gfCNCPoint2[18031] = {X 270.1696, Y 41.5937, Z -3.0000, A 0.000, B 0.000, C 0.000 }
gfCNCPoint2[18032] = {X 270.6458, Y 42.3821, Z -3.0000, A 0.000, B 0.000, C 0.000 }
gfCNCPoint2[18033] = {X 270.9441, Y 43.2536, Z -3.0000, A 0.000, B 0.000, C 0.000 }
gfCNCPoint2[18034] = {X 271.0508, Y 44.1686, Z -3.0000, A 0.000, B 0.000, C 0.000 }
gfCNCPoint2[18035] = {X 271.0510, Y 45.0000, Z -3.0000, A 0.000, B 0.000, C 0.000 }
gfCNCPoint2[18036] = {X 270.9427, Y 45.9613, Z -3.0000, A 0.000, B 0.000, C 0.000 }
gfCNCPoint2[18037] = {X 270.6232, Y 46.8744, Z -3.0000, A 0.000, B 0.000, C 0.000 }
gfCNCPoint2[18038] = {X 270.1085, Y 47.6935, Z -3.0000, A 0.000, B 0.000, C 0.000 }
gfCNCPoint2[18039] = {X 269.4245, Y 48.3775, Z -3.0000, A 0.000, B 0.000, C 0.000 }
gfCNCPoint2[18040] = {X 268.6054, Y 48.8922, Z -3.0000, A 0.000, B 0.000, C 0.000 }
gfCNCPoint2[18041] = {X 267.6923, Y 49.2117, Z -3.0000, A 0.000, B 0.000, C 0.000 }
gfCNCPoint2[18042] = {X 266.7310, Y 49.3200, Z -3.0000, A 0.000, B 0.000, C 0.000 }
gfCNCPoint2[18043] = {X 260.2876, Y 49.3200, Z -3.0000, A 0.000, B 0.000, C 0.000 }
gfCNCPoint2[18044] = {X 259.3310, Y 49.2128, Z -3.0000, A 0.000, B 0.000, C 0.000 }
gfCNCPoint2[18045] = {X 258.4219, Y 48.8963, Z -3.0000, A 0.000, B 0.000, C 0.000 }
gfCNCPoint2[18046] = {X 257.6054, Y 48.3865, Z -3.0000, A 0.000, B 0.000, C 0.000 }
gfCNCPoint2[18047] = {X 256.9221, Y 47.7085, Z -3.0000, A 0.000, B 0.000, C 0.000 }
gfCNCPoint2[18048] = {X 256.4059, Y 46.8960, Z -3.0000, A 0.000, B 0.000, C 0.000 }
gfCNCPoint2[18049] = {X 256.0824, Y 45.9894, Z -3.0000, A 0.000, B 0.000, C 0.000 }
gfCNCPoint2[18050] = {X 255.9677, Y 45.0336, Z -3.0000, A 0.000, B 0.000, C 0.000 }
gfCNCPoint2[18051] = {X 255.9680, Y 44.1494, Z -3.0000, A 0.000, B 0.000, C 0.000 }
gfCNCPoint2[18052] = {X 256.0784, Y 43.2364, Z -3.0000, A 0.000, B 0.000, C 0.000 }
gfCNCPoint2[18053] = {X 256.3796, Y 42.3675, Z -3.0000, A 0.000, B 0.000, C 0.000 }
gfCNCPoint2[18054] = {X 256.8579, Y 41.5821, Z -3.0000, A 0.000, B 0.000, C 0.000 }
gfCNCPoint2[18055] = {X 257.4915, Y 40.9157, Z -3.0000, A 0.000, B 0.000, C 0.000 }
gfCNCPoint2[18056] = {X 257.4915, Y 34.4738, Z -3.0000, A 0.000, B 0.000, C 0.000 }
gfCNCPoint2[18057] = {X 254.7671, Y 34.4738, Z -3.0000, A 0.000, B 0.000, C 0.000 }
gfCNCPoint2[18058] = {X 250.4836, Y 42.8182, Z -3.0000, A 0.000, B 0.000, C 0.000 }
gfCNCPoint2[18059] = {X 250.6527, Y 43.4861, Z -3.0000, A 0.000, B 0.000, C 0.000 }
gfCNCPoint2[18060] = {X 250.7134, Y 44.1723, Z -3.0000, A 0.000, B 0.000, C 0.000 }
gfCNCPoint2[18061] = {X 250.7136, Y 45.0000, Z -3.0000, A 0.000, B 0.000, C 0.000 }
gfCNCPoint2[18062] = {X 250.6052, Y 45.9613, Z -3.0000, A 0.000, B 0.000, C 0.000 }
gfCNCPoint2[18063] = {X 250.2857, Y 46.8744, Z -3.0000, A 0.000, B 0.000, C 0.000 }
gfCNCPoint2[18064] = {X 249.7711, Y 47.6935, Z -3.0000, A 0.000, B 0.000, C 0.000 }
gfCNCPoint2[18065] = {X 249.0870, Y 48.3775, Z -3.0000, A 0.000, B 0.000, C 0.000 }
gfCNCPoint2[18066] = {X 248.2679, Y 48.8922, Z -3.0000, A 0.000, B 0.000, C 0.000 }
gfCNCPoint2[18067] = {X 247.3548, Y 49.2117, Z -3.0000, A 0.000, B 0.000, C 0.000 }
gfCNCPoint2[18068] = {X 246.3936, Y 49.3200, Z -3.0000, A 0.000, B 0.000, C 0.000 }
gfCNCPoint2[18069] = {X 239.8075, Y 49.3200, Z -3.0000, A 0.000, B 0.000, C 0.000 }
gfCNCPoint2[18070] = {X 238.8462, Y 49.2117, Z -3.0000, A 0.000, B 0.000, C 0.000 }
gfCNCPoint2[18071] = {X 237.9331, Y 48.8922, Z -3.0000, A 0.000, B 0.000, C 0.000 }
gfCNCPoint2[18072] = {X 237.1141, Y 48.3775, Z -3.0000, A 0.000, B 0.000, C 0.000 }
gfCNCPoint2[18073] = {X 236.4300, Y 47.6935, Z -3.0000, A 0.000, B 0.000, C 0.000 }
gfCNCPoint2[18074] = {X 235.9153, Y 46.8745, Z -3.0000, A 0.000, B 0.000, C 0.000 }
gfCNCPoint2[18075] = {X 235.5958, Y 45.9614, Z -3.0000, A 0.000, B 0.000, C 0.000 }
gfCNCPoint2[18076] = {X 235.4875, Y 45.0001, Z -3.0000, A 0.000, B 0.000, C 0.000 }
gfCNCPoint2[18077] = {X 235.4879, Y 44.1494, Z -3.0000, A 0.000, B 0.000, C 0.000 }
gfCNCPoint2[18078] = {X 235.5856, Y 43.2935, Z -3.0000, A 0.000, B 0.000, C 0.000 }
gfCNCPoint2[18079] = {X 235.8511, Y 42.4740, Z -3.0000, A 0.000, B 0.000, C 0.000 }
gfCNCPoint2[18080] = {X 236.2739, Y 41.7236, Z -3.0000, A 0.000, B 0.000, C 0.000 }
gfCNCPoint2[18081] = {X 236.8373, Y 41.0719, Z -3.0000, A 0.000, B 0.000, C 0.000 }
gfCNCPoint2[18082] = {X 237.5187, Y 40.5449, Z -3.0000, A 0.000, B 0.000, C 0.000 }
gfCNCPoint2[18083] = {X 238.2911, Y 40.1637, Z -3.0000, A 0.000, B 0.000, C 0.000 }
gfCNCPoint2[18084] = {X 242.2805, Y 32.3549, Z -3.0000, A 0.000, B 0.000, C 0.000 }
gfCNCPoint2[18085] = {X 241.1106, Y 31.5686, Z -3.0000, A 0.000, B 0.000, C 0.000 }
gfCNCPoint2[18086] = {X 240.0474, Y 30.6429, Z -3.0000, A 0.000, B 0.000, C 0.000 }
gfCNCPoint2[18087] = {X 239.1077, Y 29.5922, Z -3.0000, A 0.000, B 0.000, C 0.000 }
gfCNCPoint2[18088] = {X 238.3058, Y 28.4329, Z -3.0000, A 0.000, B 0.000, C 0.000 }
gfCNCPoint2[18089] = {X 237.6543, Y 27.1828, Z -3.0000, A 0.000, B 0.000, C 0.000 }
gfCNCPoint2[18090] = {X 237.1633, Y 25.8614, Z -3.0000, A 0.000, B 0.000, C 0.000 }
gfCNCPoint2[18091] = {X 236.7431, Y 24.0500, Z -3.0000, A 0.000, B 0.000, C 0.000 }
gfCNCPoint2[18092] = {X 236.5290, Y 22.2028, Z -3.0000, A 0.000, B 0.000, C 0.000 }
gfCNCPoint2[18093] = {X 236.5236, Y 20.3432, Z -3.0000, A 0.000, B 0.000, C 0.000 }
gfCNCPoint2[18094] = {X 236.7271, Y 18.4949, Z -3.0000, A 0.000, B 0.000, C 0.000 }
gfCNCPoint2[18095] = {X 237.1368, Y 16.6810, Z -3.0000, A 0.000, B 0.000, C 0.000 }
gfCNCPoint2[18096] = {X 237.7071, Y 15.1054, Z -3.0000, A 0.000, B 0.000, C 0.000 }
gfCNCPoint2[18097] = {X 238.4940, Y 13.6260, Z -3.0000, A 0.000, B 0.000, C 0.000 }
gfCNCPoint2[18098] = {X 239.4818, Y 12.2725, Z -3.0000, A 0.000, B 0.000, C 0.000 }
gfCNCPoint2[18099] = {X 240.6507, Y 11.0718, Z -3.0000, A 0.000, B 0.000, C 0.000 }
gfCNCPoint2[18100] = {X 241.9772, Y 10.0481, Z -3.0000, A 0.000, B 0.000, C 0.000 }
gfCNCPoint2[18101] = {X 243.4350, Y 9.2218, Z -3.0000, A 0.000, B 0.000, C 0.000 }
gfCNCPoint2[18102] = {X 244.9947, Y 8.6094, Z -3.0000, A 0.000, B 0.000, C 0.000 }
gfCNCPoint2[18103] = {X 246.6252, Y 8.2232, Z -3.0000, A 0.000, B 0.000, C 0.000 }
gfCNCPoint2[18104] = {X 248.7221, Y 7.9518, Z -3.0000, A 0.000, B 0.000, C 0.000 }
gfCNCPoint2[18105] = {X 250.8350, Y 7.8712, Z -3.0000, A 0.000, B 0.000, C 0.000 }
gfCNCPoint2[18106] = {X 266.7634, Y 7.8712, Z -3.0000, A 0.000, B 0.000, C 0.000 }
gfCNCPoint2[18107] = {X 267.7184, Y 7.9860, Z -3.0000, A 0.000, B 0.000, C 0.000 }
gfCNCPoint2[18108] = {X 268.6245, Y 8.3091, Z -3.0000, A 0.000, B 0.000, C 0.000 }
gfCNCPoint2[18109] = {X 269.4366, Y 8.8247, Z -3.0000, A 0.000, B 0.000, C 0.000 }
gfCNCPoint2[18110] = {X 270.1147, Y 9.5070, Z -3.0000, A 0.000, B 0.000, C 0.000 }
gfCNCPoint2[18111] = {X 270.6250, Y 10.3225, Z -3.0000, A 0.000, B 0.000, C 0.000 }
gfCNCPoint2[18112] = {X 270.9424, Y 11.2305, Z -3.0000, A 0.000, B 0.000, C 0.000 }
gfCNCPoint2[18113] = {X 271.0510, Y 12.1863, Z -3.0000, A 0.000, B 0.000, C 0.000 }
gfCNCPoint2[18114] = {X 271.0508, Y 13.0225, Z -3.0000, A 0.000, B 0.000, C 0.000 }
gfCNCPoint2[18115] = {X 270.9424, Y 13.9406, Z -3.0000, A 0.000, B 0.000, C 0.000 }
gfCNCPoint2[18116] = {X 270.6412, Y 14.8147, Z -3.0000, A 0.000, B 0.000, C 0.000 }
gfCNCPoint2[18117] = {X 270.1608, Y 15.6046, Z -3.0000, A 0.000, B 0.000, C 0.000 }
gfCNCPoint2[18118] = {X 269.5234, Y 16.2742, Z -3.0000, A 0.000, B 0.000, C 0.000 }
gfCNCPoint2[18119] = {X 269.5233, Y 28.5936, Z -3.0000, A 0.000, B 0.000, C 0.000 }
gfCNCPoint2[18120] = {X 273.5233, Y 28.5937, Z -3.0000, A 0.000, B 0.000, C 0.000 }
gfCNCPoint2[18121] = {X 269.4433, Y 28.5936, Z -3.0000, A 0.000, B 0.000, C 0.000 }
gfCNCPoint2[18122] = {X 269.4432, Y 40.9513, Z -3.0000, A 0.000, B 0.000, C 0.000 }
gfCNCPoint2[18123] = {X 269.4859, Y 40.9857, Z -3.0000, A 0.000, B 0.000, C 0.000 }
gfCNCPoint2[18124] = {X 270.1064, Y 41.6428, Z -3.0000, A 0.000, B 0.000, C 0.000 }
gfCNCPoint2[18125] = {X 270.5736, Y 42.4165, Z -3.0000, A 0.000, B 0.000, C 0.000 }
gfCNCPoint2[18126] = {X 270.8662, Y 43.2716, Z -3.0000, A 0.000, B 0.000, C 0.000 }
gfCNCPoint2[18127] = {X 270.9708, Y 44.1693, Z -3.0000, A 0.000, B 0.000, C 0.000 }
gfCNCPoint2[18128] = {X 270.9710, Y 45.0000, Z -3.0000, A 0.000, B 0.000, C 0.000 }
gfCNCPoint2[18129] = {X 270.8647, Y 45.9435, Z -3.0000, A 0.000, B 0.000, C 0.000 }
gfCNCPoint2[18130] = {X 270.5511, Y 46.8397, Z -3.0000, A 0.000, B 0.000, C 0.000 }
gfCNCPoint2[18131] = {X 270.0460, Y 47.6436, Z -3.0000, A 0.000, B 0.000, C 0.000 }
gfCNCPoint2[18132] = {X 269.3746, Y 48.3150, Z -3.0000, A 0.000, B 0.000, C 0.000 }
gfCNCPoint2[18133] = {X 268.5707, Y 48.8201, Z -3.0000, A 0.000, B 0.000, C 0.000 }
gfCNCPoint2[18134] = {X 267.6745, Y 49.1337, Z -3.0000, A 0.000, B 0.000, C 0.000 }
gfCNCPoint2[18135] = {X 266.7310, Y 49.2400, Z -3.0000, A 0.000, B 0.000, C 0.000 }
gfCNCPoint2[18136] = {X 260.2876, Y 49.2400, Z -3.0000, A 0.000, B 0.000, C 0.000 }
gfCNCPoint2[18137] = {X 259.3487, Y 49.1347, Z -3.0000, A 0.000, B 0.000, C 0.000 }
gfCNCPoint2[18138] = {X 258.4564, Y 48.8242, Z -3.0000, A 0.000, B 0.000, C 0.000 }
gfCNCPoint2[18139] = {X 257.6550, Y 48.3238, Z -3.0000, A 0.000, B 0.000, C 0.000 }
gfCNCPoint2[18140] = {X 256.9844, Y 47.6583, Z -3.0000, A 0.000, B 0.000, C 0.000 }
gfCNCPoint2[18141] = {X 256.4777, Y 46.8609, Z -3.0000, A 0.000, B 0.000, C 0.000 }
gfCNCPoint2[18142] = {X 256.1603, Y 45.9711, Z -3.0000, A 0.000, B 0.000, C 0.000 }
gfCNCPoint2[18143] = {X 256.0477, Y 45.0330, Z -3.0000, A 0.000, B 0.000, C 0.000 }
gfCNCPoint2[18144] = {X 256.0480, Y 44.1505, Z -3.0000, A 0.000, B 0.000, C 0.000 }
gfCNCPoint2[18145] = {X 256.1585, Y 43.2454, Z -3.0000, A 0.000, B 0.000, C 0.000 }
gfCNCPoint2[18146] = {X 256.4599, Y 42.3850, Z -3.0000, A 0.000, B 0.000, C 0.000 }
gfCNCPoint2[18147] = {X 256.9383, Y 41.6088, Z -3.0000, A 0.000, B 0.000, C 0.000 }
gfCNCPoint2[18148] = {X 257.5715, Y 40.9529, Z -3.0000, A 0.000, B 0.000, C 0.000 }
gfCNCPoint2[18149] = {X 257.5715, Y 34.3938, Z -3.0000, A 0.000, B 0.000, C 0.000 }
gfCNCPoint2[18150] = {X 254.7182, Y 34.3938, Z -3.0000, A 0.000, B 0.000, C 0.000 }
gfCNCPoint2[18151] = {X 250.3969, Y 42.8120, Z -3.0000, A 0.000, B 0.000, C 0.000 }
gfCNCPoint2[18152] = {X 250.5709, Y 43.4828, Z -3.0000, A 0.000, B 0.000, C 0.000 }
gfCNCPoint2[18153] = {X 250.6334, Y 44.1730, Z -3.0000, A 0.000, B 0.000, C 0.000 }
gfCNCPoint2[18154] = {X 250.6336, Y 45.0000, Z -3.0000, A 0.000, B 0.000, C 0.000 }
gfCNCPoint2[18155] = {X 250.5273, Y 45.9435, Z -3.0000, A 0.000, B 0.000, C 0.000 }
gfCNCPoint2[18156] = {X 250.2137, Y 46.8397, Z -3.0000, A 0.000, B 0.000, C 0.000 }
gfCNCPoint2[18157] = {X 249.7085, Y 47.6436, Z -3.0000, A 0.000, B 0.000, C 0.000 }
gfCNCPoint2[18158] = {X 249.0372, Y 48.3150, Z -3.0000, A 0.000, B 0.000, C 0.000 }
gfCNCPoint2[18159] = {X 248.2332, Y 48.8201, Z -3.0000, A 0.000, B 0.000, C 0.000 }
gfCNCPoint2[18160] = {X 247.3370, Y 49.1337, Z -3.0000, A 0.000, B 0.000, C 0.000 }
gfCNCPoint2[18161] = {X 246.3936, Y 49.2400, Z -3.0000, A 0.000, B 0.000, C 0.000 }
gfCNCPoint2[18162] = {X 239.8075, Y 49.2400, Z -3.0000, A 0.000, B 0.000, C 0.000 }
gfCNCPoint2[18163] = {X 238.8640, Y 49.1337, Z -3.0000, A 0.000, B 0.000, C 0.000 }
gfCNCPoint2[18164] = {X 237.9679, Y 48.8201, Z -3.0000, A 0.000, B 0.000, C 0.000 }
gfCNCPoint2[18165] = {X 237.1639, Y 48.3150, Z -3.0000, A 0.000, B 0.000, C 0.000 }
gfCNCPoint2[18166] = {X 236.4926, Y 47.6436, Z -3.0000, A 0.000, B 0.000, C 0.000 }
gfCNCPoint2[18167] = {X 235.9874, Y 46.8397, Z -3.0000, A 0.000, B 0.000, C 0.000 }
gfCNCPoint2[18168] = {X 235.6738, Y 45.9436, Z -3.0000, A 0.000, B 0.000, C 0.000 }
gfCNCPoint2[18169] = {X 235.5675, Y 45.0001, Z -3.0000, A 0.000, B 0.000, C 0.000 }
gfCNCPoint2[18170] = {X 235.5679, Y 44.1505, Z -3.0000, A 0.000, B 0.000, C 0.000 }
gfCNCPoint2[18171] = {X 235.6649, Y 43.3054, Z -3.0000, A 0.000, B 0.000, C 0.000 }
gfCNCPoint2[18172] = {X 235.9285, Y 42.4967, Z -3.0000, A 0.000, B 0.000, C 0.000 }
gfCNCPoint2[18173] = {X 236.3483, Y 41.7570, Z -3.0000, A 0.000, B 0.000, C 0.000 }
gfCNCPoint2[18174] = {X 236.9073, Y 41.1159, Z -3.0000, A 0.000, B 0.000, C 0.000 }
gfCNCPoint2[18175] = {X 237.5830, Y 40.5992, Z -3.0000, A 0.000, B 0.000, C 0.000 }
gfCNCPoint2[18176] = {X 238.3482, Y 40.2278, Z -3.0000, A 0.000, B 0.000, C 0.000 }
gfCNCPoint2[18177] = {X 242.3863, Y 32.3238, Z -3.0000, A 0.000, B 0.000, C 0.000 }
gfCNCPoint2[18178] = {X 241.2093, Y 31.5432, Z -3.0000, A 0.000, B 0.000, C 0.000 }
gfCNCPoint2[18179] = {X 240.1396, Y 30.6212, Z -3.0000, A 0.000, B 0.000, C 0.000 }
gfCNCPoint2[18180] = {X 239.1939, Y 29.5723, Z -3.0000, A 0.000, B 0.000, C 0.000 }
gfCNCPoint2[18181] = {X 238.3873, Y 28.4131, Z -3.0000, A 0.000, B 0.000, C 0.000 }
gfCNCPoint2[18182] = {X 237.7325, Y 27.1618, Z -3.0000, A 0.000, B 0.000, C 0.000 }
gfCNCPoint2[18183] = {X 237.2398, Y 25.8383, Z -3.0000, A 0.000, B 0.000, C 0.000 }
gfCNCPoint2[18184] = {X 236.8218, Y 24.0357, Z -3.0000, A 0.000, B 0.000, C 0.000 }
gfCNCPoint2[18185] = {X 236.6088, Y 22.1976, Z -3.0000, A 0.000, B 0.000, C 0.000 }
gfCNCPoint2[18186] = {X 236.6035, Y 20.3472, Z -3.0000, A 0.000, B 0.000, C 0.000 }
gfCNCPoint2[18187] = {X 236.8060, Y 18.5079, Z -3.0000, A 0.000, B 0.000, C 0.000 }
gfCNCPoint2[18188] = {X 237.2138, Y 16.7029, Z -3.0000, A 0.000, B 0.000, C 0.000 }
gfCNCPoint2[18189] = {X 237.7802, Y 15.1379, Z -3.0000, A 0.000, B 0.000, C 0.000 }
gfCNCPoint2[18190] = {X 238.5619, Y 13.6684, Z -3.0000, A 0.000, B 0.000, C 0.000 }
gfCNCPoint2[18191] = {X 239.5430, Y 12.3240, Z -3.0000, A 0.000, B 0.000, C 0.000 }
gfCNCPoint2[18192] = {X 240.7041, Y 11.1314, Z -3.0000, A 0.000, B 0.000, C 0.000 }
gfCNCPoint2[18193] = {X 242.0217, Y 10.1146, Z -3.0000, A 0.000, B 0.000, C 0.000 }
gfCNCPoint2[18194] = {X 243.4697, Y 9.2938, Z -3.0000, A 0.000, B 0.000, C 0.000 }
gfCNCPoint2[18195] = {X 245.0190, Y 8.6856, Z -3.0000, A 0.000, B 0.000, C 0.000 }
gfCNCPoint2[18196] = {X 246.6386, Y 8.3021, Z -3.0000, A 0.000, B 0.000, C 0.000 }
gfCNCPoint2[18197] = {X 248.7287, Y 8.0315, Z -3.0000, A 0.000, B 0.000, C 0.000 }
gfCNCPoint2[18198] = {X 250.8346, Y 7.9512, Z -3.0000, A 0.000, B 0.000, C 0.000 }
gfCNCPoint2[18199] = {X 266.7627, Y 7.9512, Z -3.0000, A 0.000, B 0.000, C 0.000 }
gfCNCPoint2[18200] = {X 267.7001, Y 8.0639, Z -3.0000, A 0.000, B 0.000, C 0.000 }
gfCNCPoint2[18201] = {X 268.5894, Y 8.3810, Z -3.0000, A 0.000, B 0.000, C 0.000 }
gfCNCPoint2[18202] = {X 269.3865, Y 8.8870, Z -3.0000, A 0.000, B 0.000, C 0.000 }
gfCNCPoint2[18203] = {X 270.0520, Y 9.5568, Z -3.0000, A 0.000, B 0.000, C 0.000 }
gfCNCPoint2[18204] = {X 270.5529, Y 10.3571, Z -3.0000, A 0.000, B 0.000, C 0.000 }
gfCNCPoint2[18205] = {X 270.8644, Y 11.2484, Z -3.0000, A 0.000, B 0.000, C 0.000 }
gfCNCPoint2[18206] = {X 270.9710, Y 12.1865, Z -3.0000, A 0.000, B 0.000, C 0.000 }
gfCNCPoint2[18207] = {X 270.9708, Y 13.0217, Z -3.0000, A 0.000, B 0.000, C 0.000 }
gfCNCPoint2[18208] = {X 270.8624, Y 13.9318, Z -3.0000, A 0.000, B 0.000, C 0.000 }
gfCNCPoint2[18209] = {X 270.5609, Y 14.7973, Z -3.0000, A 0.000, B 0.000, C 0.000 }
gfCNCPoint2[18210] = {X 270.0804, Y 15.5779, Z -3.0000, A 0.000, B 0.000, C 0.000 }
gfCNCPoint2[18211] = {X 269.4434, Y 16.2369, Z -3.0000, A 0.000, B 0.000, C 0.000 }
gfCNCPoint2[18212] = {X 269.4433, Y 28.5936, Z -3.0000, A 0.000, B 0.000, C 0.000 }
gfCNCPoint2[18213] = {X 273.4433, Y 28.5937, Z -3.0000, A 0.000, B 0.000, C 0.000 }
gfCNCPoint2[18214] = {X 269.3633, Y 28.5936, Z -3.0000, A 0.000, B 0.000, C 0.000 }
gfCNCPoint2[18215] = {X 269.3632, Y 40.9896, Z -3.0000, A 0.000, B 0.000, C 0.000 }
gfCNCPoint2[18216] = {X 269.4348, Y 41.0472, Z -3.0000, A 0.000, B 0.000, C 0.000 }
gfCNCPoint2[18217] = {X 270.0432, Y 41.6919, Z -3.0000, A 0.000, B 0.000, C 0.000 }
gfCNCPoint2[18218] = {X 270.5013, Y 42.4508, Z -3.0000, A 0.000, B 0.000, C 0.000 }
gfCNCPoint2[18219] = {X 270.7882, Y 43.2896, Z -3.0000, A 0.000, B 0.000, C 0.000 }
gfCNCPoint2[18220] = {X 270.8909, Y 44.1700, Z -3.0000, A 0.000, B 0.000, C 0.000 }
gfCNCPoint2[18221] = {X 270.8910, Y 45.0000, Z -3.0000, A 0.000, B 0.000, C 0.000 }
gfCNCPoint2[18222] = {X 270.7867, Y 45.9257, Z -3.0000, A 0.000, B 0.000, C 0.000 }
gfCNCPoint2[18223] = {X 270.4791, Y 46.8050, Z -3.0000, A 0.000, B 0.000, C 0.000 }
gfCNCPoint2[18224] = {X 269.9835, Y 47.5937, Z -3.0000, A 0.000, B 0.000, C 0.000 }
gfCNCPoint2[18225] = {X 269.3247, Y 48.2524, Z -3.0000, A 0.000, B 0.000, C 0.000 }
gfCNCPoint2[18226] = {X 268.5360, Y 48.7480, Z -3.0000, A 0.000, B 0.000, C 0.000 }
gfCNCPoint2[18227] = {X 267.6567, Y 49.0557, Z -3.0000, A 0.000, B 0.000, C 0.000 }
gfCNCPoint2[18228] = {X 266.7310, Y 49.1600, Z -3.0000, A 0.000, B 0.000, C 0.000 }
gfCNCPoint2[18229] = {X 260.2876, Y 49.1600, Z -3.0000, A 0.000, B 0.000, C 0.000 }
gfCNCPoint2[18230] = {X 259.3664, Y 49.0567, Z -3.0000, A 0.000, B 0.000, C 0.000 }
gfCNCPoint2[18231] = {X 258.4910, Y 48.7520, Z -3.0000, A 0.000, B 0.000, C 0.000 }
gfCNCPoint2[18232] = {X 257.7047, Y 48.2611, Z -3.0000, A 0.000, B 0.000, C 0.000 }
gfCNCPoint2[18233] = {X 257.0467, Y 47.6082, Z -3.0000, A 0.000, B 0.000, C 0.000 }
gfCNCPoint2[18234] = {X 256.5496, Y 46.8258, Z -3.0000, A 0.000, B 0.000, C 0.000 }
gfCNCPoint2[18235] = {X 256.2381, Y 45.9527, Z -3.0000, A 0.000, B 0.000, C 0.000 }
gfCNCPoint2[18236] = {X 256.1277, Y 45.0324, Z -3.0000, A 0.000, B 0.000, C 0.000 }
gfCNCPoint2[18237] = {X 256.1280, Y 44.1516, Z -3.0000, A 0.000, B 0.000, C 0.000 }
gfCNCPoint2[18238] = {X 256.2385, Y 43.2545, Z -3.0000, A 0.000, B 0.000, C 0.000 }
gfCNCPoint2[18239] = {X 256.5401, Y 42.4026, Z -3.0000, A 0.000, B 0.000, C 0.000 }
gfCNCPoint2[18240] = {X 257.0187, Y 41.6358, Z -3.0000, A 0.000, B 0.000, C 0.000 }
gfCNCPoint2[18241] = {X 257.6515, Y 40.9906, Z -3.0000, A 0.000, B 0.000, C 0.000 }
gfCNCPoint2[18242] = {X 257.6515, Y 34.3138, Z -3.0000, A 0.000, B 0.000, C 0.000 }
gfCNCPoint2[18243] = {X 254.6694, Y 34.3138, Z -3.0000, A 0.000, B 0.000, C 0.000 }
gfCNCPoint2[18244] = {X 250.3100, Y 42.8062, Z -3.0000, A 0.000, B 0.000, C 0.000 }
gfCNCPoint2[18245] = {X 250.4892, Y 43.4797, Z -3.0000, A 0.000, B 0.000, C 0.000 }
gfCNCPoint2[18246] = {X 250.5534, Y 44.1736, Z -3.0000, A 0.000, B 0.000, C 0.000 }
gfCNCPoint2[18247] = {X 250.5536, Y 45.0000, Z -3.0000, A 0.000, B 0.000, C 0.000 }
gfCNCPoint2[18248] = {X 250.4493, Y 45.9257, Z -3.0000, A 0.000, B 0.000, C 0.000 }
gfCNCPoint2[18249] = {X 250.1416, Y 46.8050, Z -3.0000, A 0.000, B 0.000, C 0.000 }
gfCNCPoint2[18250] = {X 249.6460, Y 47.5937, Z -3.0000, A 0.000, B 0.000, C 0.000 }
gfCNCPoint2[18251] = {X 248.9873, Y 48.2524, Z -3.0000, A 0.000, B 0.000, C 0.000 }
gfCNCPoint2[18252] = {X 248.1985, Y 48.7480, Z -3.0000, A 0.000, B 0.000, C 0.000 }
gfCNCPoint2[18253] = {X 247.3192, Y 49.0557, Z -3.0000, A 0.000, B 0.000, C 0.000 }
gfCNCPoint2[18254] = {X 246.3936, Y 49.1600, Z -3.0000, A 0.000, B 0.000, C 0.000 }
gfCNCPoint2[18255] = {X 239.8075, Y 49.1600, Z -3.0000, A 0.000, B 0.000, C 0.000 }
gfCNCPoint2[18256] = {X 238.8818, Y 49.0557, Z -3.0000, A 0.000, B 0.000, C 0.000 }
gfCNCPoint2[18257] = {X 238.0026, Y 48.7480, Z -3.0000, A 0.000, B 0.000, C 0.000 }
gfCNCPoint2[18258] = {X 237.2138, Y 48.2524, Z -3.0000, A 0.000, B 0.000, C 0.000 }
gfCNCPoint2[18259] = {X 236.5551, Y 47.5937, Z -3.0000, A 0.000, B 0.000, C 0.000 }
gfCNCPoint2[18260] = {X 236.0595, Y 46.8050, Z -3.0000, A 0.000, B 0.000, C 0.000 }
gfCNCPoint2[18261] = {X 235.7518, Y 45.9257, Z -3.0000, A 0.000, B 0.000, C 0.000 }
gfCNCPoint2[18262] = {X 235.6475, Y 45.0000, Z -3.0000, A 0.000, B 0.000, C 0.000 }
gfCNCPoint2[18263] = {X 235.6479, Y 44.1516, Z -3.0000, A 0.000, B 0.000, C 0.000 }
gfCNCPoint2[18264] = {X 235.7441, Y 43.3174, Z -3.0000, A 0.000, B 0.000, C 0.000 }
gfCNCPoint2[18265] = {X 236.0059, Y 42.5195, Z -3.0000, A 0.000, B 0.000, C 0.000 }
gfCNCPoint2[18266] = {X 236.4226, Y 41.7905, Z -3.0000, A 0.000, B 0.000, C 0.000 }
gfCNCPoint2[18267] = {X 236.9772, Y 41.1600, Z -3.0000, A 0.000, B 0.000, C 0.000 }
gfCNCPoint2[18268] = {X 237.6471, Y 40.6537, Z -3.0000, A 0.000, B 0.000, C 0.000 }
gfCNCPoint2[18269] = {X 238.4051, Y 40.2923, Z -3.0000, A 0.000, B 0.000, C 0.000 }
gfCNCPoint2[18270] = {X 242.4922, Y 32.2922, Z -3.0000, A 0.000, B 0.000, C 0.000 }
gfCNCPoint2[18271] = {X 241.3082, Y 31.5176, Z -3.0000, A 0.000, B 0.000, C 0.000 }
gfCNCPoint2[18272] = {X 240.2318, Y 30.5994, Z -3.0000, A 0.000, B 0.000, C 0.000 }
gfCNCPoint2[18273] = {X 239.2803, Y 29.5524, Z -3.0000, A 0.000, B 0.000, C 0.000 }
gfCNCPoint2[18274] = {X 238.4689, Y 28.3933, Z -3.0000, A 0.000, B 0.000, C 0.000 }
gfCNCPoint2[18275] = {X 237.8108, Y 27.1408, Z -3.0000, A 0.000, B 0.000, C 0.000 }
gfCNCPoint2[18276] = {X 237.3164, Y 25.8152, Z -3.0000, A 0.000, B 0.000, C 0.000 }
gfCNCPoint2[18277] = {X 236.9005, Y 24.0214, Z -3.0000, A 0.000, B 0.000, C 0.000 }
gfCNCPoint2[18278] = {X 236.6886, Y 22.1924, Z -3.0000, A 0.000, B 0.000, C 0.000 }
gfCNCPoint2[18279] = {X 236.6834, Y 20.3511, Z -3.0000, A 0.000, B 0.000, C 0.000 }
gfCNCPoint2[18280] = {X 236.8850, Y 18.5209, Z -3.0000, A 0.000, B 0.000, C 0.000 }
gfCNCPoint2[18281] = {X 237.2907, Y 16.7248, Z -3.0000, A 0.000, B 0.000, C 0.000 }
gfCNCPoint2[18282] = {X 237.8533, Y 15.1704, Z -3.0000, A 0.000, B 0.000, C 0.000 }
gfCNCPoint2[18283] = {X 238.6297, Y 13.7108, Z -3.0000, A 0.000, B 0.000, C 0.000 }
gfCNCPoint2[18284] = {X 239.6042, Y 12.3755, Z -3.0000, A 0.000, B 0.000, C 0.000 }
gfCNCPoint2[18285] = {X 240.7574, Y 11.1910, Z -3.0000, A 0.000, B 0.000, C 0.000 }
gfCNCPoint2[18286] = {X 242.0662, Y 10.1811, Z -3.0000, A 0.000, B 0.000, C 0.000 }
gfCNCPoint2[18287] = {X 243.5045, Y 9.3659, Z -3.0000, A 0.000, B 0.000, C 0.000 }
gfCNCPoint2[18288] = {X 245.0433, Y 8.7619, Z -3.0000, A 0.000, B 0.000, C 0.000 }
gfCNCPoint2[18289] = {X 246.6520, Y 8.3810, Z -3.0000, A 0.000, B 0.000, C 0.000 }
gfCNCPoint2[18290] = {X 248.7352, Y 8.1112, Z -3.0000, A 0.000, B 0.000, C 0.000 }
gfCNCPoint2[18291] = {X 250.8343, Y 8.0312, Z -3.0000, A 0.000, B 0.000, C 0.000 }
gfCNCPoint2[18292] = {X 266.7621, Y 8.0312, Z -3.0000, A 0.000, B 0.000, C 0.000 }
gfCNCPoint2[18293] = {X 267.6818, Y 8.1418, Z -3.0000, A 0.000, B 0.000, C 0.000 }
gfCNCPoint2[18294] = {X 268.5543, Y 8.4529, Z -3.0000, A 0.000, B 0.000, C 0.000 }
gfCNCPoint2[18295] = {X 269.3364, Y 8.9494, Z -3.0000, A 0.000, B 0.000, C 0.000 }
gfCNCPoint2[18296] = {X 269.9893, Y 9.6065, Z -3.0000, A 0.000, B 0.000, C 0.000 }
gfCNCPoint2[18297] = {X 270.4808, Y 10.3917, Z -3.0000, A 0.000, B 0.000, C 0.000 }
gfCNCPoint2[18298] = {X 270.7864, Y 11.2662, Z -3.0000, A 0.000, B 0.000, C 0.000 }
gfCNCPoint2[18299] = {X 270.8910, Y 12.1866, Z -3.0000, A 0.000, B 0.000, C 0.000 }
gfCNCPoint2[18300] = {X 270.8908, Y 13.0208, Z -3.0000, A 0.000, B 0.000, C 0.000 }
gfCNCPoint2[18301] = {X 270.7823, Y 13.9229, Z -3.0000, A 0.000, B 0.000, C 0.000 }
gfCNCPoint2[18302] = {X 270.4806, Y 14.7799, Z -3.0000, A 0.000, B 0.000, C 0.000 }
gfCNCPoint2[18303] = {X 270.0000, Y 15.5509, Z -3.0000, A 0.000, B 0.000, C 0.000 }
gfCNCPoint2[18304] = {X 269.3634, Y 16.1992, Z -3.0000, A 0.000, B 0.000, C 0.000 }
gfCNCPoint2[18305] = {X 269.3633, Y 28.5936, Z -3.0000, A 0.000, B 0.000, C 0.000 }
gfCNCPoint2[18306] = {X 273.3633, Y 28.5937, Z -3.0000, A 0.000, B 0.000, C 0.000 }
gfCNCPoint2[18307] = {X 269.2833, Y 28.5936, Z -3.0000, A 0.000, B 0.000, C 0.000 }
gfCNCPoint2[18308] = {X 269.2832, Y 41.0278, Z -3.0000, A 0.000, B 0.000, C 0.000 }
gfCNCPoint2[18309] = {X 269.3836, Y 41.1088, Z -3.0000, A 0.000, B 0.000, C 0.000 }
gfCNCPoint2[18310] = {X 269.9801, Y 41.7410, Z -3.0000, A 0.000, B 0.000, C 0.000 }
gfCNCPoint2[18311] = {X 270.4291, Y 42.4851, Z -3.0000, A 0.000, B 0.000, C 0.000 }
gfCNCPoint2[18312] = {X 270.7102, Y 43.3075, Z -3.0000, A 0.000, B 0.000, C 0.000 }
gfCNCPoint2[18313] = {X 270.8109, Y 44.1708, Z -3.0000, A 0.000, B 0.000, C 0.000 }
gfCNCPoint2[18314] = {X 270.8110, Y 45.0000, Z -3.0000, A 0.000, B 0.000, C 0.000 }
gfCNCPoint2[18315] = {X 270.7087, Y 45.9079, Z -3.0000, A 0.000, B 0.000, C 0.000 }
gfCNCPoint2[18316] = {X 270.4070, Y 46.7702, Z -3.0000, A 0.000, B 0.000, C 0.000 }
gfCNCPoint2[18317] = {X 269.9209, Y 47.5438, Z -3.0000, A 0.000, B 0.000, C 0.000 }
gfCNCPoint2[18318] = {X 269.2749, Y 48.1899, Z -3.0000, A 0.000, B 0.000, C 0.000 }
gfCNCPoint2[18319] = {X 268.5013, Y 48.6760, Z -3.0000, A 0.000, B 0.000, C 0.000 }
gfCNCPoint2[18320] = {X 267.6389, Y 48.9777, Z -3.0000, A 0.000, B 0.000, C 0.000 }
gfCNCPoint2[18321] = {X 266.7310, Y 49.0800, Z -3.0000, A 0.000, B 0.000, C 0.000 }
gfCNCPoint2[18322] = {X 260.2876, Y 49.0800, Z -3.0000, A 0.000, B 0.000, C 0.000 }
gfCNCPoint2[18323] = {X 259.3841, Y 48.9787, Z -3.0000, A 0.000, B 0.000, C 0.000 }
gfCNCPoint2[18324] = {X 258.5255, Y 48.6799, Z -3.0000, A 0.000, B 0.000, C 0.000 }
gfCNCPoint2[18325] = {X 257.7544, Y 48.1983, Z -3.0000, A 0.000, B 0.000, C 0.000 }
gfCNCPoint2[18326] = {X 257.1090, Y 47.5580, Z -3.0000, A 0.000, B 0.000, C 0.000 }
gfCNCPoint2[18327] = {X 256.6215, Y 46.7907, Z -3.0000, A 0.000, B 0.000, C 0.000 }
gfCNCPoint2[18328] = {X 256.3160, Y 45.9344, Z -3.0000, A 0.000, B 0.000, C 0.000 }
gfCNCPoint2[18329] = {X 256.2077, Y 45.0318, Z -3.0000, A 0.000, B 0.000, C 0.000 }
gfCNCPoint2[18330] = {X 256.2080, Y 44.1527, Z -3.0000, A 0.000, B 0.000, C 0.000 }
gfCNCPoint2[18331] = {X 256.3185, Y 43.2637, Z -3.0000, A 0.000, B 0.000, C 0.000 }
gfCNCPoint2[18332] = {X 256.6204, Y 42.4203, Z -3.0000, A 0.000, B 0.000, C 0.000 }
gfCNCPoint2[18333] = {X 257.0991, Y 41.6631, Z -3.0000, A 0.000, B 0.000, C 0.000 }
gfCNCPoint2[18334] = {X 257.7315, Y 41.0287, Z -3.0000, A 0.000, B 0.000, C 0.000 }
gfCNCPoint2[18335] = {X 257.7315, Y 34.2338, Z -3.0000, A 0.000, B 0.000, C 0.000 }
gfCNCPoint2[18336] = {X 254.6205, Y 34.2338, Z -3.0000, A 0.000, B 0.000, C 0.000 }
gfCNCPoint2[18337] = {X 250.2229, Y 42.8007, Z -3.0000, A 0.000, B 0.000, C 0.000 }
gfCNCPoint2[18338] = {X 250.4073, Y 43.4767, Z -3.0000, A 0.000, B 0.000, C 0.000 }
gfCNCPoint2[18339] = {X 250.4734, Y 44.1743, Z -3.0000, A 0.000, B 0.000, C 0.000 }
gfCNCPoint2[18340] = {X 250.4736, Y 45.0000, Z -3.0000, A 0.000, B 0.000, C 0.000 }
gfCNCPoint2[18341] = {X 250.3713, Y 45.9079, Z -3.0000, A 0.000, B 0.000, C 0.000 }
gfCNCPoint2[18342] = {X 250.0695, Y 46.7702, Z -3.0000, A 0.000, B 0.000, C 0.000 }
gfCNCPoint2[18343] = {X 249.5834, Y 47.5438, Z -3.0000, A 0.000, B 0.000, C 0.000 }
gfCNCPoint2[18344] = {X 248.9374, Y 48.1899, Z -3.0000, A 0.000, B 0.000, C 0.000 }
gfCNCPoint2[18345] = {X 248.1638, Y 48.6760, Z -3.0000, A 0.000, B 0.000, C 0.000 }
gfCNCPoint2[18346] = {X 247.3014, Y 48.9777, Z -3.0000, A 0.000, B 0.000, C 0.000 }
gfCNCPoint2[18347] = {X 246.3936, Y 49.0800, Z -3.0000, A 0.000, B 0.000, C 0.000 }
gfCNCPoint2[18348] = {X 239.8075, Y 49.0800, Z -3.0000, A 0.000, B 0.000, C 0.000 }
gfCNCPoint2[18349] = {X 238.8996, Y 48.9777, Z -3.0000, A 0.000, B 0.000, C 0.000 }
gfCNCPoint2[18350] = {X 238.0373, Y 48.6760, Z -3.0000, A 0.000, B 0.000, C 0.000 }
gfCNCPoint2[18351] = {X 237.2637, Y 48.1899, Z -3.0000, A 0.000, B 0.000, C 0.000 }
gfCNCPoint2[18352] = {X 236.6176, Y 47.5438, Z -3.0000, A 0.000, B 0.000, C 0.000 }
gfCNCPoint2[18353] = {X 236.1315, Y 46.7702, Z -3.0000, A 0.000, B 0.000, C 0.000 }
gfCNCPoint2[18354] = {X 235.8298, Y 45.9079, Z -3.0000, A 0.000, B 0.000, C 0.000 }
gfCNCPoint2[18355] = {X 235.7275, Y 45.0000, Z -3.0000, A 0.000, B 0.000, C 0.000 }
gfCNCPoint2[18356] = {X 235.7279, Y 44.1527, Z -3.0000, A 0.000, B 0.000, C 0.000 }
gfCNCPoint2[18357] = {X 235.8234, Y 43.3294, Z -3.0000, A 0.000, B 0.000, C 0.000 }
gfCNCPoint2[18358] = {X 236.0833, Y 42.5424, Z -3.0000, A 0.000, B 0.000, C 0.000 }
gfCNCPoint2[18359] = {X 236.4969, Y 41.8242, Z -3.0000, A 0.000, B 0.000, C 0.000 }
gfCNCPoint2[18360] = {X 237.0471, Y 41.2044, Z -3.0000, A 0.000, B 0.000, C 0.000 }
gfCNCPoint2[18361] = {X 237.7112, Y 40.7085, Z -3.0000, A 0.000, B 0.000, C 0.000 }
gfCNCPoint2[18362] = {X 238.4618, Y 40.3571, Z -3.0000, A 0.000, B 0.000, C 0.000 }
gfCNCPoint2[18363] = {X 242.5984, Y 32.2602, Z -3.0000, A 0.000, B 0.000, C 0.000 }
gfCNCPoint2[18364] = {X 241.4074, Y 31.4917, Z -3.0000, A 0.000, B 0.000, C 0.000 }
gfCNCPoint2[18365] = {X 240.3242, Y 30.5774, Z -3.0000, A 0.000, B 0.000, C 0.000 }
gfCNCPoint2[18366] = {X 239.3667, Y 29.5323, Z -3.0000, A 0.000, B 0.000, C 0.000 }
gfCNCPoint2[18367] = {X 238.5505, Y 28.3734, Z -3.0000, A 0.000, B 0.000, C 0.000 }
gfCNCPoint2[18368] = {X 237.8890, Y 27.1198, Z -3.0000, A 0.000, B 0.000, C 0.000 }
gfCNCPoint2[18369] = {X 237.3930, Y 25.7920, Z -3.0000, A 0.000, B 0.000, C 0.000 }
gfCNCPoint2[18370] = {X 236.9792, Y 24.0072, Z -3.0000, A 0.000, B 0.000, C 0.000 }
gfCNCPoint2[18371] = {X 236.7685, Y 22.1872, Z -3.0000, A 0.000, B 0.000, C 0.000 }
gfCNCPoint2[18372] = {X 236.7633, Y 20.3551, Z -3.0000, A 0.000, B 0.000, C 0.000 }
gfCNCPoint2[18373] = {X 236.9639, Y 18.5339, Z -3.0000, A 0.000, B 0.000, C 0.000 }
gfCNCPoint2[18374] = {X 237.3676, Y 16.7468, Z -3.0000, A 0.000, B 0.000, C 0.000 }
gfCNCPoint2[18375] = {X 237.9264, Y 15.2029, Z -3.0000, A 0.000, B 0.000, C 0.000 }
gfCNCPoint2[18376] = {X 238.6975, Y 13.7533, Z -3.0000, A 0.000, B 0.000, C 0.000 }
gfCNCPoint2[18377] = {X 239.6654, Y 12.4270, Z -3.0000, A 0.000, B 0.000, C 0.000 }
gfCNCPoint2[18378] = {X 240.8108, Y 11.2506, Z -3.0000, A 0.000, B 0.000, C 0.000 }
gfCNCPoint2[18379] = {X 242.1107, Y 10.2475, Z -3.0000, A 0.000, B 0.000, C 0.000 }
gfCNCPoint2[18380] = {X 243.5392, Y 9.4380, Z -3.0000, A 0.000, B 0.000, C 0.000 }
gfCNCPoint2[18381] = {X 245.0676, Y 8.8381, Z -3.0000, A 0.000, B 0.000, C 0.000 }
gfCNCPoint2[18382] = {X 246.6654, Y 8.4599, Z -3.0000, A 0.000, B 0.000, C 0.000 }
gfCNCPoint2[18383] = {X 248.7417, Y 8.1910, Z -3.0000, A 0.000, B 0.000, C 0.000 }
gfCNCPoint2[18384] = {X 250.8339, Y 8.1112, Z -3.0000, A 0.000, B 0.000, C 0.000 }
gfCNCPoint2[18385] = {X 266.7614, Y 8.1112, Z -3.0000, A 0.000, B 0.000, C 0.000 }
gfCNCPoint2[18386] = {X 267.6635, Y 8.2196, Z -3.0000, A 0.000, B 0.000, C 0.000 }
gfCNCPoint2[18387] = {X 268.5192, Y 8.5248, Z -3.0000, A 0.000, B 0.000, C 0.000 }
gfCNCPoint2[18388] = {X 269.2863, Y 9.0117, Z -3.0000, A 0.000, B 0.000, C 0.000 }
gfCNCPoint2[18389] = {X 269.9267, Y 9.6562, Z -3.0000, A 0.000, B 0.000, C 0.000 }
gfCNCPoint2[18390] = {X 270.4087, Y 10.4263, Z -3.0000, A 0.000, B 0.000, C 0.000 }
gfCNCPoint2[18391] = {X 270.7084, Y 11.2840, Z -3.0000, A 0.000, B 0.000, C 0.000 }
gfCNCPoint2[18392] = {X 270.8110, Y 12.1867, Z -3.0000, A 0.000, B 0.000, C 0.000 }
gfCNCPoint2[18393] = {X 270.8108, Y 13.0200, Z -3.0000, A 0.000, B 0.000, C 0.000 }
gfCNCPoint2[18394] = {X 270.7022, Y 13.9139, Z -3.0000, A 0.000, B 0.000, C 0.000 }
gfCNCPoint2[18395] = {X 270.4002, Y 14.7622, Z -3.0000, A 0.000, B 0.000, C 0.000 }
gfCNCPoint2[18396] = {X 269.9195, Y 15.5236, Z -3.0000, A 0.000, B 0.000, C 0.000 }
gfCNCPoint2[18397] = {X 269.2834, Y 16.1610, Z -3.0000, A 0.000, B 0.000, C 0.000 }
gfCNCPoint2[18398] = {X 269.2833, Y 28.5936, Z -3.0000, A 0.000, B 0.000, C 0.000 }
gfCNCPoint2[18399] = {X 273.2833, Y 28.5937, Z -3.0000, A 0.000, B 0.000, C 0.000 }
gfCNCPoint2[18400] = {X 269.2033, Y 28.5936, Z -3.0000, A 0.000, B 0.000, C 0.000 }
gfCNCPoint2[18401] = {X 269.2032, Y 41.0661, Z -3.0000, A 0.000, B 0.000, C 0.000 }
gfCNCPoint2[18402] = {X 269.3421, Y 41.1786, Z -3.0000, A 0.000, B 0.000, C 0.000 }
gfCNCPoint2[18403] = {X 269.9283, Y 41.8051, Z -3.0000, A 0.000, B 0.000, C 0.000 }
gfCNCPoint2[18404] = {X 270.3673, Y 42.5422, Z -3.0000, A 0.000, B 0.000, C 0.000 }
gfCNCPoint2[18405] = {X 270.6391, Y 43.3559, Z -3.0000, A 0.000, B 0.000, C 0.000 }
gfCNCPoint2[18406] = {X 270.7310, Y 44.2089, Z -3.0000, A 0.000, B 0.000, C 0.000 }
gfCNCPoint2[18407] = {X 270.7310, Y 45.0000, Z -3.0000, A 0.000, B 0.000, C 0.000 }
gfCNCPoint2[18408] = {X 270.6307, Y 45.8901, Z -3.0000, A 0.000, B 0.000, C 0.000 }
gfCNCPoint2[18409] = {X 270.3349, Y 46.7355, Z -3.0000, A 0.000, B 0.000, C 0.000 }
gfCNCPoint2[18410] = {X 269.8584, Y 47.4940, Z -3.0000, A 0.000, B 0.000, C 0.000 }
gfCNCPoint2[18411] = {X 269.2250, Y 48.1273, Z -3.0000, A 0.000, B 0.000, C 0.000 }
gfCNCPoint2[18412] = {X 268.4666, Y 48.6039, Z -3.0000, A 0.000, B 0.000, C 0.000 }
gfCNCPoint2[18413] = {X 267.6211, Y 48.8997, Z -3.0000, A 0.000, B 0.000, C 0.000 }
gfCNCPoint2[18414] = {X 266.7310, Y 49.0000, Z -3.0000, A 0.000, B 0.000, C 0.000 }
gfCNCPoint2[18415] = {X 260.2876, Y 49.0000, Z -3.0000, A 0.000, B 0.000, C 0.000 }
gfCNCPoint2[18416] = {X 259.3975, Y 48.8997, Z -3.0000, A 0.000, B 0.000, C 0.000 }
gfCNCPoint2[18417] = {X 258.5520, Y 48.6039, Z -3.0000, A 0.000, B 0.000, C 0.000 }
gfCNCPoint2[18418] = {X 257.7936, Y 48.1273, Z -3.0000, A 0.000, B 0.000, C 0.000 }
gfCNCPoint2[18419] = {X 257.1602, Y 47.4939, Z -3.0000, A 0.000, B 0.000, C 0.000 }
gfCNCPoint2[18420] = {X 256.6837, Y 46.7355, Z -3.0000, A 0.000, B 0.000, C 0.000 }
gfCNCPoint2[18421] = {X 256.3878, Y 45.8900, Z -3.0000, A 0.000, B 0.000, C 0.000 }
gfCNCPoint2[18422] = {X 256.2876, Y 45.0000, Z -3.0000, A 0.000, B 0.000, C 0.000 }
gfCNCPoint2[18423] = {X 256.2879, Y 44.1538, Z -3.0000, A 0.000, B 0.000, C 0.000 }
gfCNCPoint2[18424] = {X 256.3986, Y 43.2730, Z -3.0000, A 0.000, B 0.000, C 0.000 }
gfCNCPoint2[18425] = {X 256.7008, Y 42.4382, Z -3.0000, A 0.000, B 0.000, C 0.000 }
gfCNCPoint2[18426] = {X 257.1796, Y 41.6907, Z -3.0000, A 0.000, B 0.000, C 0.000 }
gfCNCPoint2[18427] = {X 257.8115, Y 41.0672, Z -3.0000, A 0.000, B 0.000, C 0.000 }
gfCNCPoint2[18428] = {X 257.8115, Y 34.1538, Z -3.0000, A 0.000, B 0.000, C 0.000 }
gfCNCPoint2[18429] = {X 254.8159, Y 34.1538, Z -3.0000, A 0.000, B 0.000, C 0.000 }
gfCNCPoint2[18430] = {X 254.5727, Y 34.1517, Z -3.0000, A 0.000, B 0.000, C 0.000 }
gfCNCPoint2[18431] = {X 250.1356, Y 42.7956, Z -3.0000, A 0.000, B 0.000, C 0.000 }
gfCNCPoint2[18432] = {X 250.3285, Y 43.4906, Z -3.0000, A 0.000, B 0.000, C 0.000 }
gfCNCPoint2[18433] = {X 250.3936, Y 44.2089, Z -3.0000, A 0.000, B 0.000, C 0.000 }
gfCNCPoint2[18434] = {X 250.3936, Y 45.0000, Z -3.0000, A 0.000, B 0.000, C 0.000 }
gfCNCPoint2[18435] = {X 250.2933, Y 45.8901, Z -3.0000, A 0.000, B 0.000, C 0.000 }
gfCNCPoint2[18436] = {X 249.9974, Y 46.7355, Z -3.0000, A 0.000, B 0.000, C 0.000 }
gfCNCPoint2[18437] = {X 249.5209, Y 47.4940, Z -3.0000, A 0.000, B 0.000, C 0.000 }
gfCNCPoint2[18438] = {X 248.8875, Y 48.1273, Z -3.0000, A 0.000, B 0.000, C 0.000 }
gfCNCPoint2[18439] = {X 248.1291, Y 48.6039, Z -3.0000, A 0.000, B 0.000, C 0.000 }
gfCNCPoint2[18440] = {X 247.2836, Y 48.8997, Z -3.0000, A 0.000, B 0.000, C 0.000 }
gfCNCPoint2[18441] = {X 246.3936, Y 49.0000, Z -3.0000, A 0.000, B 0.000, C 0.000 }
gfCNCPoint2[18442] = {X 239.8075, Y 49.0000, Z -3.0000, A 0.000, B 0.000, C 0.000 }
gfCNCPoint2[18443] = {X 238.9174, Y 48.8997, Z -3.0000, A 0.000, B 0.000, C 0.000 }
gfCNCPoint2[18444] = {X 238.0720, Y 48.6039, Z -3.0000, A 0.000, B 0.000, C 0.000 }
gfCNCPoint2[18445] = {X 237.3135, Y 48.1273, Z -3.0000, A 0.000, B 0.000, C 0.000 }
gfCNCPoint2[18446] = {X 236.6802, Y 47.4940, Z -3.0000, A 0.000, B 0.000, C 0.000 }
gfCNCPoint2[18447] = {X 236.2036, Y 46.7355, Z -3.0000, A 0.000, B 0.000, C 0.000 }
gfCNCPoint2[18448] = {X 235.9078, Y 45.8901, Z -3.0000, A 0.000, B 0.000, C 0.000 }
gfCNCPoint2[18449] = {X 235.8075, Y 45.0000, Z -3.0000, A 0.000, B 0.000, C 0.000 }
gfCNCPoint2[18450] = {X 235.8079, Y 44.1538, Z -3.0000, A 0.000, B 0.000, C 0.000 }
gfCNCPoint2[18451] = {X 235.9027, Y 43.3414, Z -3.0000, A 0.000, B 0.000, C 0.000 }
gfCNCPoint2[18452] = {X 236.1607, Y 42.5654, Z -3.0000, A 0.000, B 0.000, C 0.000 }
gfCNCPoint2[18453] = {X 236.5712, Y 41.8580, Z -3.0000, A 0.000, B 0.000, C 0.000 }
gfCNCPoint2[18454] = {X 237.1169, Y 41.2489, Z -3.0000, A 0.000, B 0.000, C 0.000 }
gfCNCPoint2[18455] = {X 237.7752, Y 40.7635, Z -3.0000, A 0.000, B 0.000, C 0.000 }
gfCNCPoint2[18456] = {X 238.5184, Y 40.4222, Z -3.0000, A 0.000, B 0.000, C 0.000 }
gfCNCPoint2[18457] = {X 242.7049, Y 32.2276, Z -3.0000, A 0.000, B 0.000, C 0.000 }
gfCNCPoint2[18458] = {X 241.5067, Y 31.4655, Z -3.0000, A 0.000, B 0.000, C 0.000 }
gfCNCPoint2[18459] = {X 240.4168, Y 30.5552, Z -3.0000, A 0.000, B 0.000, C 0.000 }
gfCNCPoint2[18460] = {X 239.4533, Y 29.5121, Z -3.0000, A 0.000, B 0.000, C 0.000 }
gfCNCPoint2[18461] = {X 238.6322, Y 28.3535, Z -3.0000, A 0.000, B 0.000, C 0.000 }
gfCNCPoint2[18462] = {X 237.9673, Y 27.0988, Z -3.0000, A 0.000, B 0.000, C 0.000 }
gfCNCPoint2[18463] = {X 237.4696, Y 25.7689, Z -3.0000, A 0.000, B 0.000, C 0.000 }
gfCNCPoint2[18464] = {X 237.0580, Y 23.9929, Z -3.0000, A 0.000, B 0.000, C 0.000 }
gfCNCPoint2[18465] = {X 236.8483, Y 22.1820, Z -3.0000, A 0.000, B 0.000, C 0.000 }
gfCNCPoint2[18466] = {X 236.8432, Y 20.3590, Z -3.0000, A 0.000, B 0.000, C 0.000 }
gfCNCPoint2[18467] = {X 237.0428, Y 18.5469, Z -3.0000, A 0.000, B 0.000, C 0.000 }
gfCNCPoint2[18468] = {X 237.4446, Y 16.7687, Z -3.0000, A 0.000, B 0.000, C 0.000 }
gfCNCPoint2[18469] = {X 237.9995, Y 15.2354, Z -3.0000, A 0.000, B 0.000, C 0.000 }
gfCNCPoint2[18470] = {X 238.7653, Y 13.7957, Z -3.0000, A 0.000, B 0.000, C 0.000 }
gfCNCPoint2[18471] = {X 239.7266, Y 12.4785, Z -3.0000, A 0.000, B 0.000, C 0.000 }
gfCNCPoint2[18472] = {X 240.8642, Y 11.3102, Z -3.0000, A 0.000, B 0.000, C 0.000 }
gfCNCPoint2[18473] = {X 242.1552, Y 10.3140, Z -3.0000, A 0.000, B 0.000, C 0.000 }
gfCNCPoint2[18474] = {X 243.5739, Y 9.5100, Z -3.0000, A 0.000, B 0.000, C 0.000 }
gfCNCPoint2[18475] = {X 245.0919, Y 8.9143, Z -3.0000, A 0.000, B 0.000, C 0.000 }
gfCNCPoint2[18476] = {X 246.6787, Y 8.5387, Z -3.0000, A 0.000, B 0.000, C 0.000 }
gfCNCPoint2[18477] = {X 248.7483, Y 8.2707, Z -3.0000, A 0.000, B 0.000, C 0.000 }
gfCNCPoint2[18478] = {X 250.8336, Y 8.1912, Z -3.0000, A 0.000, B 0.000, C 0.000 }
gfCNCPoint2[18479] = {X 266.7608, Y 8.1912, Z -3.0000, A 0.000, B 0.000, C 0.000 }
gfCNCPoint2[18480] = {X 267.6451, Y 8.2975, Z -3.0000, A 0.000, B 0.000, C 0.000 }
gfCNCPoint2[18481] = {X 268.4841, Y 8.5967, Z -3.0000, A 0.000, B 0.000, C 0.000 }
gfCNCPoint2[18482] = {X 269.2361, Y 9.0741, Z -3.0000, A 0.000, B 0.000, C 0.000 }
gfCNCPoint2[18483] = {X 269.8640, Y 9.7059, Z -3.0000, A 0.000, B 0.000, C 0.000 }
gfCNCPoint2[18484] = {X 270.3365, Y 10.4610, Z -3.0000, A 0.000, B 0.000, C 0.000 }
gfCNCPoint2[18485] = {X 270.6304, Y 11.3018, Z -3.0000, A 0.000, B 0.000, C 0.000 }
gfCNCPoint2[18486] = {X 270.7310, Y 12.1869, Z -3.0000, A 0.000, B 0.000, C 0.000 }
gfCNCPoint2[18487] = {X 270.7308, Y 13.0192, Z -3.0000, A 0.000, B 0.000, C 0.000 }
gfCNCPoint2[18488] = {X 270.6222, Y 13.9049, Z -3.0000, A 0.000, B 0.000, C 0.000 }
gfCNCPoint2[18489] = {X 270.3199, Y 14.7444, Z -3.0000, A 0.000, B 0.000, C 0.000 }
gfCNCPoint2[18490] = {X 269.8390, Y 15.4961, Z -3.0000, A 0.000, B 0.000, C 0.000 }
gfCNCPoint2[18491] = {X 269.2034, Y 16.1224, Z -3.0000, A 0.000, B 0.000, C 0.000 }
gfCNCPoint2[18492] = {X 269.2033, Y 28.5936, Z -3.0000, A 0.000, B 0.000, C 0.000 }
gfCNCPoint2[18493] = {X 273.2833, Y 28.5937, Z -3.0000, A 0.000, B 0.000, C 0.000 }
gfCNCPoint2[18494] = {X 273.2833, Y 28.5937, Z 0.0000, A 0.000, B 0.000, C 0.000 }
gfCNCPoint2[18495] = {X 273.2833, Y 28.5937, Z 11.0000, A 0.000, B 0.000, C 0.000 }
gfCNCPoint2[18496] = {X 277.7457, Y 28.5929, Z 11.0000, A 0.000, B 0.000, C 0.000 }
gfCNCPoint2[18497] = {X 277.7457, Y 28.5929, Z 0.0000, A 0.000, B 0.000, C 0.000 }
gfCNCPoint2[18498] = {X 277.7457, Y 28.5929, Z -3.0000, A 0.000, B 0.000, C 0.000 }
gfCNCPoint2[18499] = {X 281.8257, Y 28.5928, Z -3.0000, A 0.000, B 0.000, C 0.000 }
gfCNCPoint2[18500] = {X 281.8255, Y 16.2744, Z -3.0000, A 0.000, B 0.000, C 0.000 }
gfCNCPoint2[18501] = {X 281.1869, Y 15.6033, Z -3.0000, A 0.000, B 0.000, C 0.000 }
gfCNCPoint2[18502] = {X 280.7060, Y 14.8114, Z -3.0000, A 0.000, B 0.000, C 0.000 }
gfCNCPoint2[18503] = {X 280.4051, Y 13.9353, Z -3.0000, A 0.000, B 0.000, C 0.000 }
gfCNCPoint2[18504] = {X 280.2978, Y 13.0151, Z -3.0000, A 0.000, B 0.000, C 0.000 }
gfCNCPoint2[18505] = {X 280.2977, Y 12.1868, Z -3.0000, A 0.000, B 0.000, C 0.000 }
gfCNCPoint2[18506] = {X 280.4060, Y 11.2255, Z -3.0000, A 0.000, B 0.000, C 0.000 }
gfCNCPoint2[18507] = {X 280.7255, Y 10.3124, Z -3.0000, A 0.000, B 0.000, C 0.000 }
gfCNCPoint2[18508] = {X 281.2402, Y 9.4933, Z -3.0000, A 0.000, B 0.000, C 0.000 }
gfCNCPoint2[18509] = {X 281.9242, Y 8.8093, Z -3.0000, A 0.000, B 0.000, C 0.000 }
gfCNCPoint2[18510] = {X 282.7433, Y 8.2946, Z -3.0000, A 0.000, B 0.000, C 0.000 }
gfCNCPoint2[18511] = {X 283.6564, Y 7.9751, Z -3.0000, A 0.000, B 0.000, C 0.000 }
gfCNCPoint2[18512] = {X 284.6177, Y 7.8668, Z -3.0000, A 0.000, B 0.000, C 0.000 }
gfCNCPoint2[18513] = {X 291.0611, Y 7.8668, Z -3.0000, A 0.000, B 0.000, C 0.000 }
gfCNCPoint2[18514] = {X 292.0224, Y 7.9751, Z -3.0000, A 0.000, B 0.000, C 0.000 }
gfCNCPoint2[18515] = {X 292.9355, Y 8.2946, Z -3.0000, A 0.000, B 0.000, C 0.000 }
gfCNCPoint2[18516] = {X 293.7546, Y 8.8093, Z -3.0000, A 0.000, B 0.000, C 0.000 }
gfCNCPoint2[18517] = {X 294.4386, Y 9.4933, Z -3.0000, A 0.000, B 0.000, C 0.000 }
gfCNCPoint2[18518] = {X 294.9533, Y 10.3124, Z -3.0000, A 0.000, B 0.000, C 0.000 }
gfCNCPoint2[18519] = {X 295.2728, Y 11.2255, Z -3.0000, A 0.000, B 0.000, C 0.000 }
gfCNCPoint2[18520] = {X 295.3811, Y 12.1868, Z -3.0000, A 0.000, B 0.000, C 0.000 }
gfCNCPoint2[18521] = {X 295.3811, Y 12.9781, Z -3.0000, A 0.000, B 0.000, C 0.000 }
gfCNCPoint2[18522] = {X 295.2797, Y 13.9082, Z -3.0000, A 0.000, B 0.000, C 0.000 }
gfCNCPoint2[18523] = {X 294.9804, Y 14.7947, Z -3.0000, A 0.000, B 0.000, C 0.000 }
gfCNCPoint2[18524] = {X 294.4973, Y 15.5959, Z -3.0000, A 0.000, B 0.000, C 0.000 }
gfCNCPoint2[18525] = {X 293.8530, Y 16.2743, Z -3.0000, A 0.000, B 0.000, C 0.000 }
gfCNCPoint2[18526] = {X 293.8542, Y 22.1965, Z -3.0000, A 0.000, B 0.000, C 0.000 }
gfCNCPoint2[18527] = {X 302.7596, Y 22.1965, Z -3.0000, A 0.000, B 0.000, C 0.000 }
gfCNCPoint2[18528] = {X 302.7644, Y 16.2781, Z -3.0000, A 0.000, B 0.000, C 0.000 }
gfCNCPoint2[18529] = {X 302.1243, Y 15.6070, Z -3.0000, A 0.000, B 0.000, C 0.000 }
gfCNCPoint2[18530] = {X 301.6421, Y 14.8147, Z -3.0000, A 0.000, B 0.000, C 0.000 }
gfCNCPoint2[18531] = {X 301.3402, Y 13.9377, Z -3.0000, A 0.000, B 0.000, C 0.000 }
gfCNCPoint2[18532] = {X 301.2324, Y 13.0165, Z -3.0000, A 0.000, B 0.000, C 0.000 }
gfCNCPoint2[18533] = {X 301.2323, Y 12.1868, Z -3.0000, A 0.000, B 0.000, C 0.000 }
gfCNCPoint2[18534] = {X 301.3406, Y 11.2255, Z -3.0000, A 0.000, B 0.000, C 0.000 }
gfCNCPoint2[18535] = {X 301.6601, Y 10.3124, Z -3.0000, A 0.000, B 0.000, C 0.000 }
gfCNCPoint2[18536] = {X 302.1747, Y 9.4933, Z -3.0000, A 0.000, B 0.000, C 0.000 }
gfCNCPoint2[18537] = {X 302.8588, Y 8.8093, Z -3.0000, A 0.000, B 0.000, C 0.000 }
gfCNCPoint2[18538] = {X 303.6779, Y 8.2946, Z -3.0000, A 0.000, B 0.000, C 0.000 }
gfCNCPoint2[18539] = {X 304.5910, Y 7.9751, Z -3.0000, A 0.000, B 0.000, C 0.000 }
gfCNCPoint2[18540] = {X 305.5523, Y 7.8668, Z -3.0000, A 0.000, B 0.000, C 0.000 }
gfCNCPoint2[18541] = {X 311.9957, Y 7.8668, Z -3.0000, A 0.000, B 0.000, C 0.000 }
gfCNCPoint2[18542] = {X 312.9570, Y 7.9751, Z -3.0000, A 0.000, B 0.000, C 0.000 }
gfCNCPoint2[18543] = {X 313.8701, Y 8.2946, Z -3.0000, A 0.000, B 0.000, C 0.000 }
gfCNCPoint2[18544] = {X 314.6892, Y 8.8093, Z -3.0000, A 0.000, B 0.000, C 0.000 }
gfCNCPoint2[18545] = {X 315.3732, Y 9.4933, Z -3.0000, A 0.000, B 0.000, C 0.000 }
gfCNCPoint2[18546] = {X 315.8879, Y 10.3124, Z -3.0000, A 0.000, B 0.000, C 0.000 }
gfCNCPoint2[18547] = {X 316.2074, Y 11.2255, Z -3.0000, A 0.000, B 0.000, C 0.000 }
gfCNCPoint2[18548] = {X 316.3157, Y 12.1868, Z -3.0000, A 0.000, B 0.000, C 0.000 }
gfCNCPoint2[18549] = {X 316.3157, Y 12.9781, Z -3.0000, A 0.000, B 0.000, C 0.000 }
gfCNCPoint2[18550] = {X 316.2144, Y 13.9083, Z -3.0000, A 0.000, B 0.000, C 0.000 }
gfCNCPoint2[18551] = {X 315.9151, Y 14.7948, Z -3.0000, A 0.000, B 0.000, C 0.000 }
gfCNCPoint2[18552] = {X 315.4320, Y 15.5961, Z -3.0000, A 0.000, B 0.000, C 0.000 }
gfCNCPoint2[18553] = {X 314.7877, Y 16.2745, Z -3.0000, A 0.000, B 0.000, C 0.000 }
gfCNCPoint2[18554] = {X 314.7875, Y 40.9121, Z -3.0000, A 0.000, B 0.000, C 0.000 }
gfCNCPoint2[18555] = {X 315.4262, Y 41.5831, Z -3.0000, A 0.000, B 0.000, C 0.000 }
gfCNCPoint2[18556] = {X 315.9072, Y 42.3749, Z -3.0000, A 0.000, B 0.000, C 0.000 }
gfCNCPoint2[18557] = {X 316.2082, Y 43.2511, Z -3.0000, A 0.000, B 0.000, C 0.000 }
gfCNCPoint2[18558] = {X 316.3156, Y 44.1713, Z -3.0000, A 0.000, B 0.000, C 0.000 }
gfCNCPoint2[18559] = {X 316.3157, Y 45.0000, Z -3.0000, A 0.000, B 0.000, C 0.000 }
gfCNCPoint2[18560] = {X 316.2074, Y 45.9613, Z -3.0000, A 0.000, B 0.000, C 0.000 }
gfCNCPoint2[18561] = {X 315.8879, Y 46.8744, Z -3.0000, A 0.000, B 0.000, C 0.000 }
gfCNCPoint2[18562] = {X 315.3732, Y 47.6935, Z -3.0000, A 0.000, B 0.000, C 0.000 }
gfCNCPoint2[18563] = {X 314.6892, Y 48.3775, Z -3.0000, A 0.000, B 0.000, C 0.000 }
gfCNCPoint2[18564] = {X 313.8701, Y 48.8922, Z -3.0000, A 0.000, B 0.000, C 0.000 }
gfCNCPoint2[18565] = {X 312.9570, Y 49.2117, Z -3.0000, A 0.000, B 0.000, C 0.000 }
gfCNCPoint2[18566] = {X 311.9957, Y 49.3200, Z -3.0000, A 0.000, B 0.000, C 0.000 }
gfCNCPoint2[18567] = {X 305.5523, Y 49.3200, Z -3.0000, A 0.000, B 0.000, C 0.000 }
gfCNCPoint2[18568] = {X 304.5958, Y 49.2128, Z -3.0000, A 0.000, B 0.000, C 0.000 }
gfCNCPoint2[18569] = {X 303.6868, Y 48.8965, Z -3.0000, A 0.000, B 0.000, C 0.000 }
gfCNCPoint2[18570] = {X 302.8704, Y 48.3868, Z -3.0000, A 0.000, B 0.000, C 0.000 }
gfCNCPoint2[18571] = {X 302.1872, Y 47.7090, Z -3.0000, A 0.000, B 0.000, C 0.000 }
gfCNCPoint2[18572] = {X 301.6709, Y 46.8967, Z -3.0000, A 0.000, B 0.000, C 0.000 }
gfCNCPoint2[18573] = {X 301.3473, Y 45.9903, Z -3.0000, A 0.000, B 0.000, C 0.000 }
gfCNCPoint2[18574] = {X 301.2324, Y 45.0348, Z -3.0000, A 0.000, B 0.000, C 0.000 }
gfCNCPoint2[18575] = {X 301.2323, Y 44.2011, Z -3.0000, A 0.000, B 0.000, C 0.000 }
gfCNCPoint2[18576] = {X 301.3503, Y 43.2651, Z -3.0000, A 0.000, B 0.000, C 0.000 }
gfCNCPoint2[18577] = {X 301.6537, Y 42.3717, Z -3.0000, A 0.000, B 0.000, C 0.000 }
gfCNCPoint2[18578] = {X 302.1302, Y 41.5574, Z -3.0000, A 0.000, B 0.000, C 0.000 }
gfCNCPoint2[18579] = {X 302.7604, Y 40.8554, Z -3.0000, A 0.000, B 0.000, C 0.000 }
gfCNCPoint2[18580] = {X 302.7604, Y 34.0343, Z -3.0000, A 0.000, B 0.000, C 0.000 }
gfCNCPoint2[18581] = {X 293.8540, Y 34.0343, Z -3.0000, A 0.000, B 0.000, C 0.000 }
gfCNCPoint2[18582] = {X 293.8531, Y 40.9026, Z -3.0000, A 0.000, B 0.000, C 0.000 }
gfCNCPoint2[18583] = {X 294.4921, Y 41.5866, Z -3.0000, A 0.000, B 0.000, C 0.000 }
gfCNCPoint2[18584] = {X 294.9728, Y 42.3898, Z -3.0000, A 0.000, B 0.000, C 0.000 }
gfCNCPoint2[18585] = {X 295.2737, Y 43.2762, Z -3.0000, A 0.000, B 0.000, C 0.000 }
gfCNCPoint2[18586] = {X 295.3811, Y 44.2060, Z -3.0000, A 0.000, B 0.000, C 0.000 }
gfCNCPoint2[18587] = {X 295.3811, Y 45.0000, Z -3.0000, A 0.000, B 0.000, C 0.000 }
gfCNCPoint2[18588] = {X 295.2728, Y 45.9613, Z -3.0000, A 0.000, B 0.000, C 0.000 }
gfCNCPoint2[18589] = {X 294.9533, Y 46.8744, Z -3.0000, A 0.000, B 0.000, C 0.000 }
gfCNCPoint2[18590] = {X 294.4386, Y 47.6935, Z -3.0000, A 0.000, B 0.000, C 0.000 }
gfCNCPoint2[18591] = {X 293.7546, Y 48.3775, Z -3.0000, A 0.000, B 0.000, C 0.000 }
gfCNCPoint2[18592] = {X 292.9355, Y 48.8922, Z -3.0000, A 0.000, B 0.000, C 0.000 }
gfCNCPoint2[18593] = {X 292.0224, Y 49.2117, Z -3.0000, A 0.000, B 0.000, C 0.000 }
gfCNCPoint2[18594] = {X 291.0611, Y 49.3200, Z -3.0000, A 0.000, B 0.000, C 0.000 }
gfCNCPoint2[18595] = {X 284.6177, Y 49.3200, Z -3.0000, A 0.000, B 0.000, C 0.000 }
gfCNCPoint2[18596] = {X 283.6613, Y 49.2128, Z -3.0000, A 0.000, B 0.000, C 0.000 }
gfCNCPoint2[18597] = {X 282.7524, Y 48.8965, Z -3.0000, A 0.000, B 0.000, C 0.000 }
gfCNCPoint2[18598] = {X 281.9360, Y 48.3869, Z -3.0000, A 0.000, B 0.000, C 0.000 }
gfCNCPoint2[18599] = {X 281.2527, Y 47.7092, Z -3.0000, A 0.000, B 0.000, C 0.000 }
gfCNCPoint2[18600] = {X 280.7365, Y 46.8970, Z -3.0000, A 0.000, B 0.000, C 0.000 }
gfCNCPoint2[18601] = {X 280.4128, Y 45.9907, Z -3.0000, A 0.000, B 0.000, C 0.000 }
gfCNCPoint2[18602] = {X 280.2978, Y 45.0352, Z -3.0000, A 0.000, B 0.000, C 0.000 }
gfCNCPoint2[18603] = {X 280.2977, Y 44.2071, Z -3.0000, A 0.000, B 0.000, C 0.000 }
gfCNCPoint2[18604] = {X 280.4029, Y 43.2782, Z -3.0000, A 0.000, B 0.000, C 0.000 }
gfCNCPoint2[18605] = {X 280.7032, Y 42.3929, Z -3.0000, A 0.000, B 0.000, C 0.000 }
gfCNCPoint2[18606] = {X 281.1849, Y 41.5917, Z -3.0000, A 0.000, B 0.000, C 0.000 }
gfCNCPoint2[18607] = {X 281.8259, Y 40.9112, Z -3.0000, A 0.000, B 0.000, C 0.000 }
gfCNCPoint2[18608] = {X 281.8257, Y 28.5928, Z -3.0000, A 0.000, B 0.000, C 0.000 }
gfCNCPoint2[18609] = {X 277.8257, Y 28.5929, Z -3.0000, A 0.000, B 0.000, C 0.000 }
gfCNCPoint2[18610] = {X 281.9057, Y 28.5928, Z -3.0000, A 0.000, B 0.000, C 0.000 }
gfCNCPoint2[18611] = {X 281.9055, Y 16.2371, Z -3.0000, A 0.000, B 0.000, C 0.000 }
gfCNCPoint2[18612] = {X 281.2673, Y 15.5766, Z -3.0000, A 0.000, B 0.000, C 0.000 }
gfCNCPoint2[18613] = {X 280.7863, Y 14.7942, Z -3.0000, A 0.000, B 0.000, C 0.000 }
gfCNCPoint2[18614] = {X 280.4851, Y 13.9266, Z -3.0000, A 0.000, B 0.000, C 0.000 }
gfCNCPoint2[18615] = {X 280.3778, Y 13.0144, Z -3.0000, A 0.000, B 0.000, C 0.000 }
gfCNCPoint2[18616] = {X 280.3777, Y 12.1868, Z -3.0000, A 0.000, B 0.000, C 0.000 }
gfCNCPoint2[18617] = {X 280.4840, Y 11.2433, Z -3.0000, A 0.000, B 0.000, C 0.000 }
gfCNCPoint2[18618] = {X 280.7976, Y 10.3472, Z -3.0000, A 0.000, B 0.000, C 0.000 }
gfCNCPoint2[18619] = {X 281.3027, Y 9.5432, Z -3.0000, A 0.000, B 0.000, C 0.000 }
gfCNCPoint2[18620] = {X 281.9741, Y 8.8719, Z -3.0000, A 0.000, B 0.000, C 0.000 }
gfCNCPoint2[18621] = {X 282.7780, Y 8.3667, Z -3.0000, A 0.000, B 0.000, C 0.000 }
gfCNCPoint2[18622] = {X 283.6742, Y 8.0531, Z -3.0000, A 0.000, B 0.000, C 0.000 }
gfCNCPoint2[18623] = {X 284.6177, Y 7.9468, Z -3.0000, A 0.000, B 0.000, C 0.000 }
gfCNCPoint2[18624] = {X 291.0611, Y 7.9468, Z -3.0000, A 0.000, B 0.000, C 0.000 }
gfCNCPoint2[18625] = {X 292.0046, Y 8.0531, Z -3.0000, A 0.000, B 0.000, C 0.000 }
gfCNCPoint2[18626] = {X 292.9008, Y 8.3667, Z -3.0000, A 0.000, B 0.000, C 0.000 }
gfCNCPoint2[18627] = {X 293.7047, Y 8.8718, Z -3.0000, A 0.000, B 0.000, C 0.000 }
gfCNCPoint2[18628] = {X 294.3761, Y 9.5432, Z -3.0000, A 0.000, B 0.000, C 0.000 }
gfCNCPoint2[18629] = {X 294.8812, Y 10.3471, Z -3.0000, A 0.000, B 0.000, C 0.000 }
gfCNCPoint2[18630] = {X 295.1948, Y 11.2433, Z -3.0000, A 0.000, B 0.000, C 0.000 }
gfCNCPoint2[18631] = {X 295.3011, Y 12.1868, Z -3.0000, A 0.000, B 0.000, C 0.000 }
gfCNCPoint2[18632] = {X 295.3011, Y 12.9781, Z -3.0000, A 0.000, B 0.000, C 0.000 }
gfCNCPoint2[18633] = {X 295.1996, Y 13.9000, Z -3.0000, A 0.000, B 0.000, C 0.000 }
gfCNCPoint2[18634] = {X 294.9000, Y 14.7778, Z -3.0000, A 0.000, B 0.000, C 0.000 }
gfCNCPoint2[18635] = {X 294.4168, Y 15.5694, Z -3.0000, A 0.000, B 0.000, C 0.000 }
gfCNCPoint2[18636] = {X 293.7730, Y 16.2370, Z -3.0000, A 0.000, B 0.000, C 0.000 }
gfCNCPoint2[18637] = {X 293.7742, Y 22.2765, Z -3.0000, A 0.000, B 0.000, C 0.000 }
gfCNCPoint2[18638] = {X 302.8396, Y 22.2765, Z -3.0000, A 0.000, B 0.000, C 0.000 }
gfCNCPoint2[18639] = {X 302.8445, Y 16.2408, Z -3.0000, A 0.000, B 0.000, C 0.000 }
gfCNCPoint2[18640] = {X 302.2047, Y 15.5803, Z -3.0000, A 0.000, B 0.000, C 0.000 }
gfCNCPoint2[18641] = {X 301.7225, Y 14.7974, Z -3.0000, A 0.000, B 0.000, C 0.000 }
gfCNCPoint2[18642] = {X 301.4203, Y 13.9290, Z -3.0000, A 0.000, B 0.000, C 0.000 }
gfCNCPoint2[18643] = {X 301.3124, Y 13.0158, Z -3.0000, A 0.000, B 0.000, C 0.000 }
gfCNCPoint2[18644] = {X 301.3123, Y 12.1868, Z -3.0000, A 0.000, B 0.000, C 0.000 }
gfCNCPoint2[18645] = {X 301.4186, Y 11.2433, Z -3.0000, A 0.000, B 0.000, C 0.000 }
gfCNCPoint2[18646] = {X 301.7321, Y 10.3471, Z -3.0000, A 0.000, B 0.000, C 0.000 }
gfCNCPoint2[18647] = {X 302.2373, Y 9.5432, Z -3.0000, A 0.000, B 0.000, C 0.000 }
gfCNCPoint2[18648] = {X 302.9087, Y 8.8718, Z -3.0000, A 0.000, B 0.000, C 0.000 }
gfCNCPoint2[18649] = {X 303.7126, Y 8.3667, Z -3.0000, A 0.000, B 0.000, C 0.000 }
gfCNCPoint2[18650] = {X 304.6088, Y 8.0531, Z -3.0000, A 0.000, B 0.000, C 0.000 }
gfCNCPoint2[18651] = {X 305.5523, Y 7.9468, Z -3.0000, A 0.000, B 0.000, C 0.000 }
gfCNCPoint2[18652] = {X 311.9957, Y 7.9468, Z -3.0000, A 0.000, B 0.000, C 0.000 }
gfCNCPoint2[18653] = {X 312.9392, Y 8.0531, Z -3.0000, A 0.000, B 0.000, C 0.000 }
gfCNCPoint2[18654] = {X 313.8354, Y 8.3667, Z -3.0000, A 0.000, B 0.000, C 0.000 }
gfCNCPoint2[18655] = {X 314.6393, Y 8.8718, Z -3.0000, A 0.000, B 0.000, C 0.000 }
gfCNCPoint2[18656] = {X 315.3107, Y 9.5432, Z -3.0000, A 0.000, B 0.000, C 0.000 }
gfCNCPoint2[18657] = {X 315.8158, Y 10.3471, Z -3.0000, A 0.000, B 0.000, C 0.000 }
gfCNCPoint2[18658] = {X 316.1294, Y 11.2433, Z -3.0000, A 0.000, B 0.000, C 0.000 }
gfCNCPoint2[18659] = {X 316.2357, Y 12.1868, Z -3.0000, A 0.000, B 0.000, C 0.000 }
gfCNCPoint2[18660] = {X 316.2357, Y 12.9781, Z -3.0000, A 0.000, B 0.000, C 0.000 }
gfCNCPoint2[18661] = {X 316.1343, Y 13.9001, Z -3.0000, A 0.000, B 0.000, C 0.000 }
gfCNCPoint2[18662] = {X 315.8347, Y 14.7779, Z -3.0000, A 0.000, B 0.000, C 0.000 }
gfCNCPoint2[18663] = {X 315.3515, Y 15.5696, Z -3.0000, A 0.000, B 0.000, C 0.000 }
gfCNCPoint2[18664] = {X 314.7077, Y 16.2372, Z -3.0000, A 0.000, B 0.000, C 0.000 }
gfCNCPoint2[18665] = {X 314.7075, Y 40.9506, Z -3.0000, A 0.000, B 0.000, C 0.000 }
gfCNCPoint2[18666] = {X 314.7358, Y 40.9731, Z -3.0000, A 0.000, B 0.000, C 0.000 }
gfCNCPoint2[18667] = {X 315.3627, Y 41.6317, Z -3.0000, A 0.000, B 0.000, C 0.000 }
gfCNCPoint2[18668] = {X 315.8347, Y 42.4089, Z -3.0000, A 0.000, B 0.000, C 0.000 }
gfCNCPoint2[18669] = {X 316.1302, Y 43.2688, Z -3.0000, A 0.000, B 0.000, C 0.000 }
gfCNCPoint2[18670] = {X 316.2356, Y 44.1720, Z -3.0000, A 0.000, B 0.000, C 0.000 }
gfCNCPoint2[18671] = {X 316.2357, Y 45.0000, Z -3.0000, A 0.000, B 0.000, C 0.000 }
gfCNCPoint2[18672] = {X 316.1294, Y 45.9435, Z -3.0000, A 0.000, B 0.000, C 0.000 }
gfCNCPoint2[18673] = {X 315.8158, Y 46.8397, Z -3.0000, A 0.000, B 0.000, C 0.000 }
gfCNCPoint2[18674] = {X 315.3107, Y 47.6436, Z -3.0000, A 0.000, B 0.000, C 0.000 }
gfCNCPoint2[18675] = {X 314.6393, Y 48.3150, Z -3.0000, A 0.000, B 0.000, C 0.000 }
gfCNCPoint2[18676] = {X 313.8354, Y 48.8201, Z -3.0000, A 0.000, B 0.000, C 0.000 }
gfCNCPoint2[18677] = {X 312.9392, Y 49.1337, Z -3.0000, A 0.000, B 0.000, C 0.000 }
gfCNCPoint2[18678] = {X 311.9957, Y 49.2400, Z -3.0000, A 0.000, B 0.000, C 0.000 }
gfCNCPoint2[18679] = {X 305.5523, Y 49.2400, Z -3.0000, A 0.000, B 0.000, C 0.000 }
gfCNCPoint2[18680] = {X 304.6135, Y 49.1348, Z -3.0000, A 0.000, B 0.000, C 0.000 }
gfCNCPoint2[18681] = {X 303.7214, Y 48.8243, Z -3.0000, A 0.000, B 0.000, C 0.000 }
gfCNCPoint2[18682] = {X 302.9201, Y 48.3241, Z -3.0000, A 0.000, B 0.000, C 0.000 }
gfCNCPoint2[18683] = {X 302.2495, Y 47.6588, Z -3.0000, A 0.000, B 0.000, C 0.000 }
gfCNCPoint2[18684] = {X 301.7428, Y 46.8616, Z -3.0000, A 0.000, B 0.000, C 0.000 }
gfCNCPoint2[18685] = {X 301.4252, Y 45.9720, Z -3.0000, A 0.000, B 0.000, C 0.000 }
gfCNCPoint2[18686] = {X 301.3124, Y 45.0341, Z -3.0000, A 0.000, B 0.000, C 0.000 }
gfCNCPoint2[18687] = {X 301.3123, Y 44.2031, Z -3.0000, A 0.000, B 0.000, C 0.000 }
gfCNCPoint2[18688] = {X 301.4302, Y 43.2744, Z -3.0000, A 0.000, B 0.000, C 0.000 }
gfCNCPoint2[18689] = {X 301.7338, Y 42.3889, Z -3.0000, A 0.000, B 0.000, C 0.000 }
gfCNCPoint2[18690] = {X 302.2104, Y 41.5833, Z -3.0000, A 0.000, B 0.000, C 0.000 }
gfCNCPoint2[18691] = {X 302.8404, Y 40.8909, Z -3.0000, A 0.000, B 0.000, C 0.000 }
gfCNCPoint2[18692] = {X 302.8404, Y 33.9543, Z -3.0000, A 0.000, B 0.000, C 0.000 }
gfCNCPoint2[18693] = {X 293.7740, Y 33.9543, Z -3.0000, A 0.000, B 0.000, C 0.000 }
gfCNCPoint2[18694] = {X 293.7731, Y 40.9394, Z -3.0000, A 0.000, B 0.000, C 0.000 }
gfCNCPoint2[18695] = {X 294.4117, Y 41.6129, Z -3.0000, A 0.000, B 0.000, C 0.000 }
gfCNCPoint2[18696] = {X 294.8925, Y 42.4068, Z -3.0000, A 0.000, B 0.000, C 0.000 }
gfCNCPoint2[18697] = {X 295.1936, Y 43.2848, Z -3.0000, A 0.000, B 0.000, C 0.000 }
gfCNCPoint2[18698] = {X 295.3011, Y 44.2067, Z -3.0000, A 0.000, B 0.000, C 0.000 }
gfCNCPoint2[18699] = {X 295.3011, Y 45.0000, Z -3.0000, A 0.000, B 0.000, C 0.000 }
gfCNCPoint2[18700] = {X 295.1948, Y 45.9435, Z -3.0000, A 0.000, B 0.000, C 0.000 }
gfCNCPoint2[18701] = {X 294.8812, Y 46.8397, Z -3.0000, A 0.000, B 0.000, C 0.000 }
gfCNCPoint2[18702] = {X 294.3761, Y 47.6436, Z -3.0000, A 0.000, B 0.000, C 0.000 }
gfCNCPoint2[18703] = {X 293.7047, Y 48.3150, Z -3.0000, A 0.000, B 0.000, C 0.000 }
gfCNCPoint2[18704] = {X 292.9008, Y 48.8201, Z -3.0000, A 0.000, B 0.000, C 0.000 }
gfCNCPoint2[18705] = {X 292.0046, Y 49.1337, Z -3.0000, A 0.000, B 0.000, C 0.000 }
gfCNCPoint2[18706] = {X 291.0611, Y 49.2400, Z -3.0000, A 0.000, B 0.000, C 0.000 }
gfCNCPoint2[18707] = {X 284.6177, Y 49.2400, Z -3.0000, A 0.000, B 0.000, C 0.000 }
gfCNCPoint2[18708] = {X 283.6790, Y 49.1348, Z -3.0000, A 0.000, B 0.000, C 0.000 }
gfCNCPoint2[18709] = {X 282.7869, Y 48.8244, Z -3.0000, A 0.000, B 0.000, C 0.000 }
gfCNCPoint2[18710] = {X 281.9857, Y 48.3242, Z -3.0000, A 0.000, B 0.000, C 0.000 }
gfCNCPoint2[18711] = {X 281.3150, Y 47.6590, Z -3.0000, A 0.000, B 0.000, C 0.000 }
gfCNCPoint2[18712] = {X 280.8083, Y 46.8619, Z -3.0000, A 0.000, B 0.000, C 0.000 }
gfCNCPoint2[18713] = {X 280.4907, Y 45.9723, Z -3.0000, A 0.000, B 0.000, C 0.000 }
gfCNCPoint2[18714] = {X 280.3778, Y 45.0345, Z -3.0000, A 0.000, B 0.000, C 0.000 }
gfCNCPoint2[18715] = {X 280.3777, Y 44.2075, Z -3.0000, A 0.000, B 0.000, C 0.000 }
gfCNCPoint2[18716] = {X 280.4830, Y 43.2867, Z -3.0000, A 0.000, B 0.000, C 0.000 }
gfCNCPoint2[18717] = {X 280.7835, Y 42.4099, Z -3.0000, A 0.000, B 0.000, C 0.000 }
gfCNCPoint2[18718] = {X 281.2653, Y 41.6181, Z -3.0000, A 0.000, B 0.000, C 0.000 }
gfCNCPoint2[18719] = {X 281.9059, Y 40.9482, Z -3.0000, A 0.000, B 0.000, C 0.000 }
gfCNCPoint2[18720] = {X 281.9057, Y 28.5928, Z -3.0000, A 0.000, B 0.000, C 0.000 }
gfCNCPoint2[18721] = {X 277.9057, Y 28.5929, Z -3.0000, A 0.000, B 0.000, C 0.000 }
gfCNCPoint2[18722] = {X 281.9857, Y 28.5928, Z -3.0000, A 0.000, B 0.000, C 0.000 }
gfCNCPoint2[18723] = {X 281.9855, Y 16.1994, Z -3.0000, A 0.000, B 0.000, C 0.000 }
gfCNCPoint2[18724] = {X 281.3478, Y 15.5497, Z -3.0000, A 0.000, B 0.000, C 0.000 }
gfCNCPoint2[18725] = {X 280.8667, Y 14.7768, Z -3.0000, A 0.000, B 0.000, C 0.000 }
gfCNCPoint2[18726] = {X 280.5652, Y 13.9178, Z -3.0000, A 0.000, B 0.000, C 0.000 }
gfCNCPoint2[18727] = {X 280.4578, Y 13.0137, Z -3.0000, A 0.000, B 0.000, C 0.000 }
gfCNCPoint2[18728] = {X 280.4577, Y 12.1868, Z -3.0000, A 0.000, B 0.000, C 0.000 }
gfCNCPoint2[18729] = {X 280.5620, Y 11.2611, Z -3.0000, A 0.000, B 0.000, C 0.000 }
gfCNCPoint2[18730] = {X 280.8696, Y 10.3819, Z -3.0000, A 0.000, B 0.000, C 0.000 }
gfCNCPoint2[18731] = {X 281.3652, Y 9.5931, Z -3.0000, A 0.000, B 0.000, C 0.000 }
gfCNCPoint2[18732] = {X 282.0240, Y 8.9344, Z -3.0000, A 0.000, B 0.000, C 0.000 }
gfCNCPoint2[18733] = {X 282.8127, Y 8.4388, Z -3.0000, A 0.000, B 0.000, C 0.000 }
gfCNCPoint2[18734] = {X 283.6920, Y 8.1311, Z -3.0000, A 0.000, B 0.000, C 0.000 }
gfCNCPoint2[18735] = {X 284.6177, Y 8.0268, Z -3.0000, A 0.000, B 0.000, C 0.000 }
gfCNCPoint2[18736] = {X 291.0611, Y 8.0268, Z -3.0000, A 0.000, B 0.000, C 0.000 }
gfCNCPoint2[18737] = {X 291.9868, Y 8.1311, Z -3.0000, A 0.000, B 0.000, C 0.000 }
gfCNCPoint2[18738] = {X 292.8661, Y 8.4388, Z -3.0000, A 0.000, B 0.000, C 0.000 }
gfCNCPoint2[18739] = {X 293.6549, Y 8.9344, Z -3.0000, A 0.000, B 0.000, C 0.000 }
gfCNCPoint2[18740] = {X 294.3136, Y 9.5931, Z -3.0000, A 0.000, B 0.000, C 0.000 }
gfCNCPoint2[18741] = {X 294.8092, Y 10.3819, Z -3.0000, A 0.000, B 0.000, C 0.000 }
gfCNCPoint2[18742] = {X 295.1168, Y 11.2611, Z -3.0000, A 0.000, B 0.000, C 0.000 }
gfCNCPoint2[18743] = {X 295.2211, Y 12.1868, Z -3.0000, A 0.000, B 0.000, C 0.000 }
gfCNCPoint2[18744] = {X 295.2211, Y 12.9781, Z -3.0000, A 0.000, B 0.000, C 0.000 }
gfCNCPoint2[18745] = {X 295.1254, Y 13.8653, Z -3.0000, A 0.000, B 0.000, C 0.000 }
gfCNCPoint2[18746] = {X 294.8427, Y 14.7116, Z -3.0000, A 0.000, B 0.000, C 0.000 }
gfCNCPoint2[18747] = {X 294.3860, Y 15.4782, Z -3.0000, A 0.000, B 0.000, C 0.000 }
gfCNCPoint2[18748] = {X 293.7763, Y 16.1297, Z -3.0000, A 0.000, B 0.000, C 0.000 }
gfCNCPoint2[18749] = {X 293.6930, Y 16.1997, Z -3.0000, A 0.000, B 0.000, C 0.000 }
gfCNCPoint2[18750] = {X 293.6943, Y 22.3567, Z -3.0000, A 0.000, B 0.000, C 0.000 }
gfCNCPoint2[18751] = {X 302.9195, Y 22.3565, Z -3.0000, A 0.000, B 0.000, C 0.000 }
gfCNCPoint2[18752] = {X 302.9245, Y 16.2030, Z -3.0000, A 0.000, B 0.000, C 0.000 }
gfCNCPoint2[18753] = {X 302.2852, Y 15.5533, Z -3.0000, A 0.000, B 0.000, C 0.000 }
gfCNCPoint2[18754] = {X 301.8028, Y 14.7800, Z -3.0000, A 0.000, B 0.000, C 0.000 }
gfCNCPoint2[18755] = {X 301.5003, Y 13.9202, Z -3.0000, A 0.000, B 0.000, C 0.000 }
gfCNCPoint2[18756] = {X 301.3924, Y 13.0151, Z -3.0000, A 0.000, B 0.000, C 0.000 }
gfCNCPoint2[18757] = {X 301.3923, Y 12.1868, Z -3.0000, A 0.000, B 0.000, C 0.000 }
gfCNCPoint2[18758] = {X 301.4966, Y 11.2611, Z -3.0000, A 0.000, B 0.000, C 0.000 }
gfCNCPoint2[18759] = {X 301.8042, Y 10.3819, Z -3.0000, A 0.000, B 0.000, C 0.000 }
gfCNCPoint2[18760] = {X 302.2998, Y 9.5931, Z -3.0000, A 0.000, B 0.000, C 0.000 }
gfCNCPoint2[18761] = {X 302.9585, Y 8.9344, Z -3.0000, A 0.000, B 0.000, C 0.000 }
gfCNCPoint2[18762] = {X 303.7473, Y 8.4388, Z -3.0000, A 0.000, B 0.000, C 0.000 }
gfCNCPoint2[18763] = {X 304.6266, Y 8.1311, Z -3.0000, A 0.000, B 0.000, C 0.000 }
gfCNCPoint2[18764] = {X 305.5523, Y 8.0268, Z -3.0000, A 0.000, B 0.000, C 0.000 }
gfCNCPoint2[18765] = {X 311.9957, Y 8.0268, Z -3.0000, A 0.000, B 0.000, C 0.000 }
gfCNCPoint2[18766] = {X 312.9214, Y 8.1311, Z -3.0000, A 0.000, B 0.000, C 0.000 }
gfCNCPoint2[18767] = {X 313.8007, Y 8.4388, Z -3.0000, A 0.000, B 0.000, C 0.000 }
gfCNCPoint2[18768] = {X 314.5894, Y 8.9344, Z -3.0000, A 0.000, B 0.000, C 0.000 }
gfCNCPoint2[18769] = {X 315.2481, Y 9.5931, Z -3.0000, A 0.000, B 0.000, C 0.000 }
gfCNCPoint2[18770] = {X 315.7438, Y 10.3819, Z -3.0000, A 0.000, B 0.000, C 0.000 }
gfCNCPoint2[18771] = {X 316.0514, Y 11.2611, Z -3.0000, A 0.000, B 0.000, C 0.000 }
gfCNCPoint2[18772] = {X 316.1557, Y 12.1868, Z -3.0000, A 0.000, B 0.000, C 0.000 }
gfCNCPoint2[18773] = {X 316.1557, Y 12.9781, Z -3.0000, A 0.000, B 0.000, C 0.000 }
gfCNCPoint2[18774] = {X 316.0542, Y 13.8916, Z -3.0000, A 0.000, B 0.000, C 0.000 }
gfCNCPoint2[18775] = {X 315.7545, Y 14.7605, Z -3.0000, A 0.000, B 0.000, C 0.000 }
gfCNCPoint2[18776] = {X 315.2713, Y 15.5424, Z -3.0000, A 0.000, B 0.000, C 0.000 }
gfCNCPoint2[18777] = {X 314.6283, Y 16.1991, Z -3.0000, A 0.000, B 0.000, C 0.000 }
gfCNCPoint2[18778] = {X 314.6275, Y 40.9893, Z -3.0000, A 0.000, B 0.000, C 0.000 }
gfCNCPoint2[18779] = {X 314.6833, Y 41.0335, Z -3.0000, A 0.000, B 0.000, C 0.000 }
gfCNCPoint2[18780] = {X 315.2987, Y 41.6797, Z -3.0000, A 0.000, B 0.000, C 0.000 }
gfCNCPoint2[18781] = {X 315.7621, Y 42.4424, Z -3.0000, A 0.000, B 0.000, C 0.000 }
gfCNCPoint2[18782] = {X 316.0521, Y 43.2863, Z -3.0000, A 0.000, B 0.000, C 0.000 }
gfCNCPoint2[18783] = {X 316.1556, Y 44.1727, Z -3.0000, A 0.000, B 0.000, C 0.000 }
gfCNCPoint2[18784] = {X 316.1557, Y 45.0000, Z -3.0000, A 0.000, B 0.000, C 0.000 }
gfCNCPoint2[18785] = {X 316.0514, Y 45.9257, Z -3.0000, A 0.000, B 0.000, C 0.000 }
gfCNCPoint2[18786] = {X 315.7438, Y 46.8050, Z -3.0000, A 0.000, B 0.000, C 0.000 }
gfCNCPoint2[18787] = {X 315.2481, Y 47.5937, Z -3.0000, A 0.000, B 0.000, C 0.000 }
gfCNCPoint2[18788] = {X 314.5894, Y 48.2524, Z -3.0000, A 0.000, B 0.000, C 0.000 }
gfCNCPoint2[18789] = {X 313.8007, Y 48.7480, Z -3.0000, A 0.000, B 0.000, C 0.000 }
gfCNCPoint2[18790] = {X 312.9214, Y 49.0557, Z -3.0000, A 0.000, B 0.000, C 0.000 }
gfCNCPoint2[18791] = {X 311.9957, Y 49.1600, Z -3.0000, A 0.000, B 0.000, C 0.000 }
gfCNCPoint2[18792] = {X 305.5523, Y 49.1600, Z -3.0000, A 0.000, B 0.000, C 0.000 }
gfCNCPoint2[18793] = {X 304.6312, Y 49.0568, Z -3.0000, A 0.000, B 0.000, C 0.000 }
gfCNCPoint2[18794] = {X 303.7559, Y 48.7522, Z -3.0000, A 0.000, B 0.000, C 0.000 }
gfCNCPoint2[18795] = {X 302.9698, Y 48.2613, Z -3.0000, A 0.000, B 0.000, C 0.000 }
gfCNCPoint2[18796] = {X 302.3118, Y 47.6087, Z -3.0000, A 0.000, B 0.000, C 0.000 }
gfCNCPoint2[18797] = {X 301.8147, Y 46.8265, Z -3.0000, A 0.000, B 0.000, C 0.000 }
gfCNCPoint2[18798] = {X 301.5030, Y 45.9537, Z -3.0000, A 0.000, B 0.000, C 0.000 }
gfCNCPoint2[18799] = {X 301.3924, Y 45.0335, Z -3.0000, A 0.000, B 0.000, C 0.000 }
gfCNCPoint2[18800] = {X 301.3923, Y 44.2050, Z -3.0000, A 0.000, B 0.000, C 0.000 }
gfCNCPoint2[18801] = {X 301.5102, Y 43.2839, Z -3.0000, A 0.000, B 0.000, C 0.000 }
gfCNCPoint2[18802] = {X 301.8139, Y 42.4063, Z -3.0000, A 0.000, B 0.000, C 0.000 }
gfCNCPoint2[18803] = {X 302.2907, Y 41.6094, Z -3.0000, A 0.000, B 0.000, C 0.000 }
gfCNCPoint2[18804] = {X 302.9204, Y 40.9268, Z -3.0000, A 0.000, B 0.000, C 0.000 }
gfCNCPoint2[18805] = {X 302.9204, Y 33.8743, Z -3.0000, A 0.000, B 0.000, C 0.000 }
gfCNCPoint2[18806] = {X 293.6940, Y 33.8743, Z -3.0000, A 0.000, B 0.000, C 0.000 }
gfCNCPoint2[18807] = {X 293.6931, Y 40.9766, Z -3.0000, A 0.000, B 0.000, C 0.000 }
gfCNCPoint2[18808] = {X 294.3313, Y 41.6395, Z -3.0000, A 0.000, B 0.000, C 0.000 }
gfCNCPoint2[18809] = {X 294.8122, Y 42.4241, Z -3.0000, A 0.000, B 0.000, C 0.000 }
gfCNCPoint2[18810] = {X 295.1135, Y 43.2936, Z -3.0000, A 0.000, B 0.000, C 0.000 }
gfCNCPoint2[18811] = {X 295.2211, Y 44.2075, Z -3.0000, A 0.000, B 0.000, C 0.000 }
gfCNCPoint2[18812] = {X 295.2211, Y 45.0000, Z -3.0000, A 0.000, B 0.000, C 0.000 }
gfCNCPoint2[18813] = {X 295.1168, Y 45.9257, Z -3.0000, A 0.000, B 0.000, C 0.000 }
gfCNCPoint2[18814] = {X 294.8092, Y 46.8050, Z -3.0000, A 0.000, B 0.000, C 0.000 }
gfCNCPoint2[18815] = {X 294.3136, Y 47.5937, Z -3.0000, A 0.000, B 0.000, C 0.000 }
gfCNCPoint2[18816] = {X 293.6549, Y 48.2524, Z -3.0000, A 0.000, B 0.000, C 0.000 }
gfCNCPoint2[18817] = {X 292.8661, Y 48.7480, Z -3.0000, A 0.000, B 0.000, C 0.000 }
gfCNCPoint2[18818] = {X 291.9868, Y 49.0557, Z -3.0000, A 0.000, B 0.000, C 0.000 }
gfCNCPoint2[18819] = {X 291.0611, Y 49.1600, Z -3.0000, A 0.000, B 0.000, C 0.000 }
gfCNCPoint2[18820] = {X 284.6177, Y 49.1600, Z -3.0000, A 0.000, B 0.000, C 0.000 }
gfCNCPoint2[18821] = {X 283.6967, Y 49.0568, Z -3.0000, A 0.000, B 0.000, C 0.000 }
gfCNCPoint2[18822] = {X 282.8214, Y 48.7522, Z -3.0000, A 0.000, B 0.000, C 0.000 }
gfCNCPoint2[18823] = {X 282.0353, Y 48.2615, Z -3.0000, A 0.000, B 0.000, C 0.000 }
gfCNCPoint2[18824] = {X 281.3774, Y 47.6088, Z -3.0000, A 0.000, B 0.000, C 0.000 }
gfCNCPoint2[18825] = {X 280.8802, Y 46.8267, Z -3.0000, A 0.000, B 0.000, C 0.000 }
gfCNCPoint2[18826] = {X 280.5685, Y 45.9540, Z -3.0000, A 0.000, B 0.000, C 0.000 }
gfCNCPoint2[18827] = {X 280.4578, Y 45.0339, Z -3.0000, A 0.000, B 0.000, C 0.000 }
gfCNCPoint2[18828] = {X 280.4577, Y 44.2080, Z -3.0000, A 0.000, B 0.000, C 0.000 }
gfCNCPoint2[18829] = {X 280.5631, Y 43.2952, Z -3.0000, A 0.000, B 0.000, C 0.000 }
gfCNCPoint2[18830] = {X 280.8639, Y 42.4271, Z -3.0000, A 0.000, B 0.000, C 0.000 }
gfCNCPoint2[18831] = {X 281.3458, Y 41.6448, Z -3.0000, A 0.000, B 0.000, C 0.000 }
gfCNCPoint2[18832] = {X 281.9859, Y 40.9857, Z -3.0000, A 0.000, B 0.000, C 0.000 }
gfCNCPoint2[18833] = {X 281.9857, Y 28.5928, Z -3.0000, A 0.000, B 0.000, C 0.000 }
gfCNCPoint2[18834] = {X 277.9857, Y 28.5929, Z -3.0000, A 0.000, B 0.000, C 0.000 }
gfCNCPoint2[18835] = {X 282.0657, Y 28.5928, Z -3.0000, A 0.000, B 0.000, C 0.000 }
gfCNCPoint2[18836] = {X 282.0655, Y 16.1612, Z -3.0000, A 0.000, B 0.000, C 0.000 }
gfCNCPoint2[18837] = {X 281.4283, Y 15.5225, Z -3.0000, A 0.000, B 0.000, C 0.000 }
gfCNCPoint2[18838] = {X 280.9470, Y 14.7592, Z -3.0000, A 0.000, B 0.000, C 0.000 }
gfCNCPoint2[18839] = {X 280.6453, Y 13.9089, Z -3.0000, A 0.000, B 0.000, C 0.000 }
gfCNCPoint2[18840] = {X 280.5378, Y 13.0130, Z -3.0000, A 0.000, B 0.000, C 0.000 }
gfCNCPoint2[18841] = {X 280.5377, Y 12.1868, Z -3.0000, A 0.000, B 0.000, C 0.000 }
gfCNCPoint2[18842] = {X 280.6400, Y 11.2789, Z -3.0000, A 0.000, B 0.000, C 0.000 }
gfCNCPoint2[18843] = {X 280.9417, Y 10.4166, Z -3.0000, A 0.000, B 0.000, C 0.000 }
gfCNCPoint2[18844] = {X 281.4278, Y 9.6430, Z -3.0000, A 0.000, B 0.000, C 0.000 }
gfCNCPoint2[18845] = {X 282.0738, Y 8.9969, Z -3.0000, A 0.000, B 0.000, C 0.000 }
gfCNCPoint2[18846] = {X 282.8474, Y 8.5109, Z -3.0000, A 0.000, B 0.000, C 0.000 }
gfCNCPoint2[18847] = {X 283.7098, Y 8.2091, Z -3.0000, A 0.000, B 0.000, C 0.000 }
gfCNCPoint2[18848] = {X 284.6177, Y 8.1068, Z -3.0000, A 0.000, B 0.000, C 0.000 }
gfCNCPoint2[18849] = {X 291.0611, Y 8.1068, Z -3.0000, A 0.000, B 0.000, C 0.000 }
gfCNCPoint2[18850] = {X 291.9690, Y 8.2091, Z -3.0000, A 0.000, B 0.000, C 0.000 }
gfCNCPoint2[18851] = {X 292.8314, Y 8.5109, Z -3.0000, A 0.000, B 0.000, C 0.000 }
gfCNCPoint2[18852] = {X 293.6050, Y 8.9969, Z -3.0000, A 0.000, B 0.000, C 0.000 }
gfCNCPoint2[18853] = {X 294.2510, Y 9.6430, Z -3.0000, A 0.000, B 0.000, C 0.000 }
gfCNCPoint2[18854] = {X 294.7371, Y 10.4166, Z -3.0000, A 0.000, B 0.000, C 0.000 }
gfCNCPoint2[18855] = {X 295.0388, Y 11.2789, Z -3.0000, A 0.000, B 0.000, C 0.000 }
gfCNCPoint2[18856] = {X 295.1411, Y 12.1868, Z -3.0000, A 0.000, B 0.000, C 0.000 }
gfCNCPoint2[18857] = {X 295.1411, Y 12.9781, Z -3.0000, A 0.000, B 0.000, C 0.000 }
gfCNCPoint2[18858] = {X 295.0473, Y 13.8482, Z -3.0000, A 0.000, B 0.000, C 0.000 }
gfCNCPoint2[18859] = {X 294.7700, Y 14.6783, Z -3.0000, A 0.000, B 0.000, C 0.000 }
gfCNCPoint2[18860] = {X 294.3221, Y 15.4301, Z -3.0000, A 0.000, B 0.000, C 0.000 }
gfCNCPoint2[18861] = {X 293.7241, Y 16.0691, Z -3.0000, A 0.000, B 0.000, C 0.000 }
gfCNCPoint2[18862] = {X 293.6668, Y 16.1176, Z -3.0000, A 0.000, B 0.000, C 0.000 }
gfCNCPoint2[18863] = {X 293.6085, Y 16.1650, Z -3.0000, A 0.000, B 0.000, C 0.000 }
gfCNCPoint2[18864] = {X 293.6130, Y 16.1997, Z -3.0000, A 0.000, B 0.000, C 0.000 }
gfCNCPoint2[18865] = {X 293.6143, Y 22.4369, Z -3.0000, A 0.000, B 0.000, C 0.000 }
gfCNCPoint2[18866] = {X 293.7675, Y 22.4365, Z -3.0000, A 0.000, B 0.000, C 0.000 }
gfCNCPoint2[18867] = {X 302.9994, Y 22.4365, Z -3.0000, A 0.000, B 0.000, C 0.000 }
gfCNCPoint2[18868] = {X 303.0045, Y 16.1648, Z -3.0000, A 0.000, B 0.000, C 0.000 }
gfCNCPoint2[18869] = {X 302.9463, Y 16.1173, Z -3.0000, A 0.000, B 0.000, C 0.000 }
gfCNCPoint2[18870] = {X 302.8889, Y 16.0688, Z -3.0000, A 0.000, B 0.000, C 0.000 }
gfCNCPoint2[18871] = {X 302.2966, Y 15.4371, Z -3.0000, A 0.000, B 0.000, C 0.000 }
gfCNCPoint2[18872] = {X 301.8509, Y 14.6945, Z -3.0000, A 0.000, B 0.000, C 0.000 }
gfCNCPoint2[18873] = {X 301.5720, Y 13.8747, Z -3.0000, A 0.000, B 0.000, C 0.000 }
gfCNCPoint2[18874] = {X 301.4724, Y 13.0144, Z -3.0000, A 0.000, B 0.000, C 0.000 }
gfCNCPoint2[18875] = {X 301.4723, Y 12.1868, Z -3.0000, A 0.000, B 0.000, C 0.000 }
gfCNCPoint2[18876] = {X 301.5745, Y 11.2789, Z -3.0000, A 0.000, B 0.000, C 0.000 }
gfCNCPoint2[18877] = {X 301.8763, Y 10.4166, Z -3.0000, A 0.000, B 0.000, C 0.000 }
gfCNCPoint2[18878] = {X 302.3624, Y 9.6430, Z -3.0000, A 0.000, B 0.000, C 0.000 }
gfCNCPoint2[18879] = {X 303.0084, Y 8.9969, Z -3.0000, A 0.000, B 0.000, C 0.000 }
gfCNCPoint2[18880] = {X 303.7820, Y 8.5109, Z -3.0000, A 0.000, B 0.000, C 0.000 }
gfCNCPoint2[18881] = {X 304.6444, Y 8.2091, Z -3.0000, A 0.000, B 0.000, C 0.000 }
gfCNCPoint2[18882] = {X 305.5523, Y 8.1068, Z -3.0000, A 0.000, B 0.000, C 0.000 }
gfCNCPoint2[18883] = {X 311.9957, Y 8.1068, Z -3.0000, A 0.000, B 0.000, C 0.000 }
gfCNCPoint2[18884] = {X 312.9036, Y 8.2091, Z -3.0000, A 0.000, B 0.000, C 0.000 }
gfCNCPoint2[18885] = {X 313.7660, Y 8.5109, Z -3.0000, A 0.000, B 0.000, C 0.000 }
gfCNCPoint2[18886] = {X 314.5396, Y 8.9969, Z -3.0000, A 0.000, B 0.000, C 0.000 }
gfCNCPoint2[18887] = {X 315.1856, Y 9.6430, Z -3.0000, A 0.000, B 0.000, C 0.000 }
gfCNCPoint2[18888] = {X 315.6717, Y 10.4166, Z -3.0000, A 0.000, B 0.000, C 0.000 }
gfCNCPoint2[18889] = {X 315.9734, Y 11.2789, Z -3.0000, A 0.000, B 0.000, C 0.000 }
gfCNCPoint2[18890] = {X 316.0757, Y 12.1868, Z -3.0000, A 0.000, B 0.000, C 0.000 }
gfCNCPoint2[18891] = {X 316.0757, Y 12.9781, Z -3.0000, A 0.000, B 0.000, C 0.000 }
gfCNCPoint2[18892] = {X 315.9819, Y 13.8482, Z -3.0000, A 0.000, B 0.000, C 0.000 }
gfCNCPoint2[18893] = {X 315.7046, Y 14.6782, Z -3.0000, A 0.000, B 0.000, C 0.000 }
gfCNCPoint2[18894] = {X 315.2567, Y 15.4300, Z -3.0000, A 0.000, B 0.000, C 0.000 }
gfCNCPoint2[18895] = {X 314.6589, Y 16.0690, Z -3.0000, A 0.000, B 0.000, C 0.000 }
gfCNCPoint2[18896] = {X 314.6043, Y 16.1152, Z -3.0000, A 0.000, B 0.000, C 0.000 }
gfCNCPoint2[18897] = {X 314.5489, Y 16.1604, Z -3.0000, A 0.000, B 0.000, C 0.000 }
gfCNCPoint2[18898] = {X 314.5475, Y 41.0280, Z -3.0000, A 0.000, B 0.000, C 0.000 }
gfCNCPoint2[18899] = {X 314.6336, Y 41.0962, Z -3.0000, A 0.000, B 0.000, C 0.000 }
gfCNCPoint2[18900] = {X 315.2363, Y 41.7299, Z -3.0000, A 0.000, B 0.000, C 0.000 }
gfCNCPoint2[18901] = {X 315.6902, Y 42.4775, Z -3.0000, A 0.000, B 0.000, C 0.000 }
gfCNCPoint2[18902] = {X 315.9743, Y 43.3047, Z -3.0000, A 0.000, B 0.000, C 0.000 }
gfCNCPoint2[18903] = {X 316.0756, Y 44.1734, Z -3.0000, A 0.000, B 0.000, C 0.000 }
gfCNCPoint2[18904] = {X 316.0757, Y 45.0000, Z -3.0000, A 0.000, B 0.000, C 0.000 }
gfCNCPoint2[18905] = {X 315.9734, Y 45.9079, Z -3.0000, A 0.000, B 0.000, C 0.000 }
gfCNCPoint2[18906] = {X 315.6717, Y 46.7702, Z -3.0000, A 0.000, B 0.000, C 0.000 }
gfCNCPoint2[18907] = {X 315.1856, Y 47.5438, Z -3.0000, A 0.000, B 0.000, C 0.000 }
gfCNCPoint2[18908] = {X 314.5396, Y 48.1899, Z -3.0000, A 0.000, B 0.000, C 0.000 }
gfCNCPoint2[18909] = {X 313.7660, Y 48.6760, Z -3.0000, A 0.000, B 0.000, C 0.000 }
gfCNCPoint2[18910] = {X 312.9036, Y 48.9777, Z -3.0000, A 0.000, B 0.000, C 0.000 }
gfCNCPoint2[18911] = {X 311.9957, Y 49.0800, Z -3.0000, A 0.000, B 0.000, C 0.000 }
gfCNCPoint2[18912] = {X 305.5523, Y 49.0800, Z -3.0000, A 0.000, B 0.000, C 0.000 }
gfCNCPoint2[18913] = {X 304.6489, Y 48.9787, Z -3.0000, A 0.000, B 0.000, C 0.000 }
gfCNCPoint2[18914] = {X 303.7905, Y 48.6800, Z -3.0000, A 0.000, B 0.000, C 0.000 }
gfCNCPoint2[18915] = {X 303.0194, Y 48.1986, Z -3.0000, A 0.000, B 0.000, C 0.000 }
gfCNCPoint2[18916] = {X 302.3741, Y 47.5585, Z -3.0000, A 0.000, B 0.000, C 0.000 }
gfCNCPoint2[18917] = {X 301.8865, Y 46.7914, Z -3.0000, A 0.000, B 0.000, C 0.000 }
gfCNCPoint2[18918] = {X 301.5809, Y 45.9353, Z -3.0000, A 0.000, B 0.000, C 0.000 }
gfCNCPoint2[18919] = {X 301.4724, Y 45.0328, Z -3.0000, A 0.000, B 0.000, C 0.000 }
gfCNCPoint2[18920] = {X 301.4723, Y 44.2070, Z -3.0000, A 0.000, B 0.000, C 0.000 }
gfCNCPoint2[18921] = {X 301.5901, Y 43.2934, Z -3.0000, A 0.000, B 0.000, C 0.000 }
gfCNCPoint2[18922] = {X 301.8941, Y 42.4238, Z -3.0000, A 0.000, B 0.000, C 0.000 }
gfCNCPoint2[18923] = {X 302.3710, Y 41.6358, Z -3.0000, A 0.000, B 0.000, C 0.000 }
gfCNCPoint2[18924] = {X 303.0004, Y 40.9632, Z -3.0000, A 0.000, B 0.000, C 0.000 }
gfCNCPoint2[18925] = {X 303.0004, Y 33.7943, Z -3.0000, A 0.000, B 0.000, C 0.000 }
gfCNCPoint2[18926] = {X 293.6140, Y 33.7943, Z -3.0000, A 0.000, B 0.000, C 0.000 }
gfCNCPoint2[18927] = {X 293.6130, Y 41.0142, Z -3.0000, A 0.000, B 0.000, C 0.000 }
gfCNCPoint2[18928] = {X 294.2508, Y 41.6664, Z -3.0000, A 0.000, B 0.000, C 0.000 }
gfCNCPoint2[18929] = {X 294.7319, Y 42.4414, Z -3.0000, A 0.000, B 0.000, C 0.000 }
gfCNCPoint2[18930] = {X 295.0335, Y 43.3024, Z -3.0000, A 0.000, B 0.000, C 0.000 }
gfCNCPoint2[18931] = {X 295.1411, Y 44.2082, Z -3.0000, A 0.000, B 0.000, C 0.000 }
gfCNCPoint2[18932] = {X 295.1411, Y 45.0000, Z -3.0000, A 0.000, B 0.000, C 0.000 }
gfCNCPoint2[18933] = {X 295.0388, Y 45.9079, Z -3.0000, A 0.000, B 0.000, C 0.000 }
gfCNCPoint2[18934] = {X 294.7371, Y 46.7702, Z -3.0000, A 0.000, B 0.000, C 0.000 }
gfCNCPoint2[18935] = {X 294.2510, Y 47.5438, Z -3.0000, A 0.000, B 0.000, C 0.000 }
gfCNCPoint2[18936] = {X 293.6050, Y 48.1899, Z -3.0000, A 0.000, B 0.000, C 0.000 }
gfCNCPoint2[18937] = {X 292.8314, Y 48.6760, Z -3.0000, A 0.000, B 0.000, C 0.000 }
gfCNCPoint2[18938] = {X 291.9690, Y 48.9777, Z -3.0000, A 0.000, B 0.000, C 0.000 }
gfCNCPoint2[18939] = {X 291.0611, Y 49.0800, Z -3.0000, A 0.000, B 0.000, C 0.000 }
gfCNCPoint2[18940] = {X 284.6177, Y 49.0800, Z -3.0000, A 0.000, B 0.000, C 0.000 }
gfCNCPoint2[18941] = {X 283.7144, Y 48.9788, Z -3.0000, A 0.000, B 0.000, C 0.000 }
gfCNCPoint2[18942] = {X 282.8560, Y 48.6801, Z -3.0000, A 0.000, B 0.000, C 0.000 }
gfCNCPoint2[18943] = {X 282.0850, Y 48.1987, Z -3.0000, A 0.000, B 0.000, C 0.000 }
gfCNCPoint2[18944] = {X 281.4397, Y 47.5587, Z -3.0000, A 0.000, B 0.000, C 0.000 }
gfCNCPoint2[18945] = {X 280.9521, Y 46.7916, Z -3.0000, A 0.000, B 0.000, C 0.000 }
gfCNCPoint2[18946] = {X 280.6464, Y 45.9356, Z -3.0000, A 0.000, B 0.000, C 0.000 }
gfCNCPoint2[18947] = {X 280.5378, Y 45.0332, Z -3.0000, A 0.000, B 0.000, C 0.000 }
gfCNCPoint2[18948] = {X 280.5377, Y 44.2084, Z -3.0000, A 0.000, B 0.000, C 0.000 }
gfCNCPoint2[18949] = {X 280.6431, Y 43.3039, Z -3.0000, A 0.000, B 0.000, C 0.000 }
gfCNCPoint2[18950] = {X 280.9442, Y 42.4444, Z -3.0000, A 0.000, B 0.000, C 0.000 }
gfCNCPoint2[18951] = {X 281.4263, Y 41.6718, Z -3.0000, A 0.000, B 0.000, C 0.000 }
gfCNCPoint2[18952] = {X 282.0659, Y 41.0236, Z -3.0000, A 0.000, B 0.000, C 0.000 }
gfCNCPoint2[18953] = {X 282.0657, Y 28.5928, Z -3.0000, A 0.000, B 0.000, C 0.000 }
gfCNCPoint2[18954] = {X 278.0657, Y 28.5929, Z -3.0000, A 0.000, B 0.000, C 0.000 }
gfCNCPoint2[18955] = {X 282.1457, Y 28.5928, Z -3.0000, A 0.000, B 0.000, C 0.000 }
gfCNCPoint2[18956] = {X 282.1455, Y 16.1226, Z -3.0000, A 0.000, B 0.000, C 0.000 }
gfCNCPoint2[18957] = {X 281.5034, Y 15.4882, Z -3.0000, A 0.000, B 0.000, C 0.000 }
gfCNCPoint2[18958] = {X 281.0198, Y 14.7260, Z -3.0000, A 0.000, B 0.000, C 0.000 }
gfCNCPoint2[18959] = {X 280.7195, Y 13.8748, Z -3.0000, A 0.000, B 0.000, C 0.000 }
gfCNCPoint2[18960] = {X 280.6177, Y 12.9779, Z -3.0000, A 0.000, B 0.000, C 0.000 }
gfCNCPoint2[18961] = {X 280.6177, Y 12.1868, Z -3.0000, A 0.000, B 0.000, C 0.000 }
gfCNCPoint2[18962] = {X 280.7180, Y 11.2967, Z -3.0000, A 0.000, B 0.000, C 0.000 }
gfCNCPoint2[18963] = {X 281.0138, Y 10.4513, Z -3.0000, A 0.000, B 0.000, C 0.000 }
gfCNCPoint2[18964] = {X 281.4903, Y 9.6929, Z -3.0000, A 0.000, B 0.000, C 0.000 }
gfCNCPoint2[18965] = {X 282.1237, Y 9.0595, Z -3.0000, A 0.000, B 0.000, C 0.000 }
gfCNCPoint2[18966] = {X 282.8821, Y 8.5829, Z -3.0000, A 0.000, B 0.000, C 0.000 }
gfCNCPoint2[18967] = {X 283.7276, Y 8.2871, Z -3.0000, A 0.000, B 0.000, C 0.000 }
gfCNCPoint2[18968] = {X 284.6177, Y 8.1868, Z -3.0000, A 0.000, B 0.000, C 0.000 }
gfCNCPoint2[18969] = {X 291.0611, Y 8.1868, Z -3.0000, A 0.000, B 0.000, C 0.000 }
gfCNCPoint2[18970] = {X 291.9512, Y 8.2871, Z -3.0000, A 0.000, B 0.000, C 0.000 }
gfCNCPoint2[18971] = {X 292.7967, Y 8.5829, Z -3.0000, A 0.000, B 0.000, C 0.000 }
gfCNCPoint2[18972] = {X 293.5551, Y 9.0595, Z -3.0000, A 0.000, B 0.000, C 0.000 }
gfCNCPoint2[18973] = {X 294.1885, Y 9.6929, Z -3.0000, A 0.000, B 0.000, C 0.000 }
gfCNCPoint2[18974] = {X 294.6650, Y 10.4513, Z -3.0000, A 0.000, B 0.000, C 0.000 }
gfCNCPoint2[18975] = {X 294.9608, Y 11.2967, Z -3.0000, A 0.000, B 0.000, C 0.000 }
gfCNCPoint2[18976] = {X 295.0611, Y 12.1868, Z -3.0000, A 0.000, B 0.000, C 0.000 }
gfCNCPoint2[18977] = {X 295.0609, Y 13.0192, Z -3.0000, A 0.000, B 0.000, C 0.000 }
gfCNCPoint2[18978] = {X 294.9624, Y 13.8612, Z -3.0000, A 0.000, B 0.000, C 0.000 }
gfCNCPoint2[18979] = {X 294.6887, Y 14.6636, Z -3.0000, A 0.000, B 0.000, C 0.000 }
gfCNCPoint2[18980] = {X 294.2519, Y 15.3902, Z -3.0000, A 0.000, B 0.000, C 0.000 }
gfCNCPoint2[18981] = {X 293.6719, Y 16.0085, Z -3.0000, A 0.000, B 0.000, C 0.000 }
gfCNCPoint2[18982] = {X 293.5956, Y 16.0726, Z -3.0000, A 0.000, B 0.000, C 0.000 }
gfCNCPoint2[18983] = {X 293.5177, Y 16.1348, Z -3.0000, A 0.000, B 0.000, C 0.000 }
gfCNCPoint2[18984] = {X 293.5330, Y 16.1921, Z -3.0000, A 0.000, B 0.000, C 0.000 }
gfCNCPoint2[18985] = {X 293.5343, Y 22.5171, Z -3.0000, A 0.000, B 0.000, C 0.000 }
gfCNCPoint2[18986] = {X 293.7676, Y 22.5165, Z -3.0000, A 0.000, B 0.000, C 0.000 }
gfCNCPoint2[18987] = {X 303.0794, Y 22.5175, Z -3.0000, A 0.000, B 0.000, C 0.000 }
gfCNCPoint2[18988] = {X 303.0800, Y 16.1922, Z -3.0000, A 0.000, B 0.000, C 0.000 }
gfCNCPoint2[18989] = {X 303.0955, Y 16.1346, Z -3.0000, A 0.000, B 0.000, C 0.000 }
gfCNCPoint2[18990] = {X 303.0175, Y 16.0724, Z -3.0000, A 0.000, B 0.000, C 0.000 }
gfCNCPoint2[18991] = {X 302.9411, Y 16.0082, Z -3.0000, A 0.000, B 0.000, C 0.000 }
gfCNCPoint2[18992] = {X 302.3550, Y 15.3817, Z -3.0000, A 0.000, B 0.000, C 0.000 }
gfCNCPoint2[18993] = {X 301.9160, Y 14.6446, Z -3.0000, A 0.000, B 0.000, C 0.000 }
gfCNCPoint2[18994] = {X 301.6442, Y 13.8309, Z -3.0000, A 0.000, B 0.000, C 0.000 }
gfCNCPoint2[18995] = {X 301.5523, Y 12.9779, Z -3.0000, A 0.000, B 0.000, C 0.000 }
gfCNCPoint2[18996] = {X 301.5523, Y 12.1868, Z -3.0000, A 0.000, B 0.000, C 0.000 }
gfCNCPoint2[18997] = {X 301.6525, Y 11.2967, Z -3.0000, A 0.000, B 0.000, C 0.000 }
gfCNCPoint2[18998] = {X 301.9484, Y 10.4513, Z -3.0000, A 0.000, B 0.000, C 0.000 }
gfCNCPoint2[18999] = {X 302.4249, Y 9.6929, Z -3.0000, A 0.000, B 0.000, C 0.000 }
gfCNCPoint2[19000] = {X 303.0583, Y 9.0595, Z -3.0000, A 0.000, B 0.000, C 0.000 }
gfCNCPoint2[19001] = {X 303.8167, Y 8.5829, Z -3.0000, A 0.000, B 0.000, C 0.000 }
gfCNCPoint2[19002] = {X 304.6622, Y 8.2871, Z -3.0000, A 0.000, B 0.000, C 0.000 }
gfCNCPoint2[19003] = {X 305.5523, Y 8.1868, Z -3.0000, A 0.000, B 0.000, C 0.000 }
gfCNCPoint2[19004] = {X 311.9957, Y 8.1868, Z -3.0000, A 0.000, B 0.000, C 0.000 }
gfCNCPoint2[19005] = {X 312.8858, Y 8.2871, Z -3.0000, A 0.000, B 0.000, C 0.000 }
gfCNCPoint2[19006] = {X 313.7313, Y 8.5829, Z -3.0000, A 0.000, B 0.000, C 0.000 }
gfCNCPoint2[19007] = {X 314.4897, Y 9.0595, Z -3.0000, A 0.000, B 0.000, C 0.000 }
gfCNCPoint2[19008] = {X 315.1230, Y 9.6929, Z -3.0000, A 0.000, B 0.000, C 0.000 }
gfCNCPoint2[19009] = {X 315.5996, Y 10.4513, Z -3.0000, A 0.000, B 0.000, C 0.000 }
gfCNCPoint2[19010] = {X 315.8954, Y 11.2967, Z -3.0000, A 0.000, B 0.000, C 0.000 }
gfCNCPoint2[19011] = {X 315.9957, Y 12.1868, Z -3.0000, A 0.000, B 0.000, C 0.000 }
gfCNCPoint2[19012] = {X 315.9955, Y 13.0192, Z -3.0000, A 0.000, B 0.000, C 0.000 }
gfCNCPoint2[19013] = {X 315.8970, Y 13.8612, Z -3.0000, A 0.000, B 0.000, C 0.000 }
gfCNCPoint2[19014] = {X 315.6233, Y 14.6635, Z -3.0000, A 0.000, B 0.000, C 0.000 }
gfCNCPoint2[19015] = {X 315.1866, Y 15.3901, Z -3.0000, A 0.000, B 0.000, C 0.000 }
gfCNCPoint2[19016] = {X 314.6066, Y 16.0084, Z -3.0000, A 0.000, B 0.000, C 0.000 }
gfCNCPoint2[19017] = {X 314.5387, Y 16.0656, Z -3.0000, A 0.000, B 0.000, C 0.000 }
gfCNCPoint2[19018] = {X 314.4695, Y 16.1213, Z -3.0000, A 0.000, B 0.000, C 0.000 }
gfCNCPoint2[19019] = {X 314.4677, Y 16.3114, Z -3.0000, A 0.000, B 0.000, C 0.000 }
gfCNCPoint2[19020] = {X 314.4675, Y 41.0667, Z -3.0000, A 0.000, B 0.000, C 0.000 }
gfCNCPoint2[19021] = {X 314.6064, Y 41.1782, Z -3.0000, A 0.000, B 0.000, C 0.000 }
gfCNCPoint2[19022] = {X 315.1927, Y 41.8048, Z -3.0000, A 0.000, B 0.000, C 0.000 }
gfCNCPoint2[19023] = {X 315.6319, Y 42.5419, Z -3.0000, A 0.000, B 0.000, C 0.000 }
gfCNCPoint2[19024] = {X 315.9037, Y 43.3558, Z -3.0000, A 0.000, B 0.000, C 0.000 }
gfCNCPoint2[19025] = {X 315.9957, Y 44.2089, Z -3.0000, A 0.000, B 0.000, C 0.000 }
gfCNCPoint2[19026] = {X 315.9957, Y 45.0000, Z -3.0000, A 0.000, B 0.000, C 0.000 }
gfCNCPoint2[19027] = {X 315.8954, Y 45.8901, Z -3.0000, A 0.000, B 0.000, C 0.000 }
gfCNCPoint2[19028] = {X 315.5996, Y 46.7355, Z -3.0000, A 0.000, B 0.000, C 0.000 }
gfCNCPoint2[19029] = {X 315.1230, Y 47.4940, Z -3.0000, A 0.000, B 0.000, C 0.000 }
gfCNCPoint2[19030] = {X 314.4897, Y 48.1273, Z -3.0000, A 0.000, B 0.000, C 0.000 }
gfCNCPoint2[19031] = {X 313.7313, Y 48.6039, Z -3.0000, A 0.000, B 0.000, C 0.000 }
gfCNCPoint2[19032] = {X 312.8858, Y 48.8997, Z -3.0000, A 0.000, B 0.000, C 0.000 }
gfCNCPoint2[19033] = {X 311.9957, Y 49.0000, Z -3.0000, A 0.000, B 0.000, C 0.000 }
gfCNCPoint2[19034] = {X 305.5523, Y 49.0000, Z -3.0000, A 0.000, B 0.000, C 0.000 }
gfCNCPoint2[19035] = {X 304.6622, Y 48.8997, Z -3.0000, A 0.000, B 0.000, C 0.000 }
gfCNCPoint2[19036] = {X 303.8167, Y 48.6039, Z -3.0000, A 0.000, B 0.000, C 0.000 }
gfCNCPoint2[19037] = {X 303.0583, Y 48.1273, Z -3.0000, A 0.000, B 0.000, C 0.000 }
gfCNCPoint2[19038] = {X 302.4249, Y 47.4939, Z -3.0000, A 0.000, B 0.000, C 0.000 }
gfCNCPoint2[19039] = {X 301.9484, Y 46.7355, Z -3.0000, A 0.000, B 0.000, C 0.000 }
gfCNCPoint2[19040] = {X 301.6525, Y 45.8900, Z -3.0000, A 0.000, B 0.000, C 0.000 }
gfCNCPoint2[19041] = {X 301.5523, Y 45.0000, Z -3.0000, A 0.000, B 0.000, C 0.000 }
gfCNCPoint2[19042] = {X 301.5523, Y 44.2089, Z -3.0000, A 0.000, B 0.000, C 0.000 }
gfCNCPoint2[19043] = {X 301.6701, Y 43.3029, Z -3.0000, A 0.000, B 0.000, C 0.000 }
gfCNCPoint2[19044] = {X 301.9742, Y 42.4415, Z -3.0000, A 0.000, B 0.000, C 0.000 }
gfCNCPoint2[19045] = {X 302.4513, Y 41.6624, Z -3.0000, A 0.000, B 0.000, C 0.000 }
gfCNCPoint2[19046] = {X 303.0804, Y 40.9999, Z -3.0000, A 0.000, B 0.000, C 0.000 }
gfCNCPoint2[19047] = {X 303.0804, Y 33.7143, Z -3.0000, A 0.000, B 0.000, C 0.000 }
gfCNCPoint2[19048] = {X 293.9340, Y 33.7143, Z -3.0000, A 0.000, B 0.000, C 0.000 }
gfCNCPoint2[19049] = {X 293.5340, Y 33.7134, Z -3.0000, A 0.000, B 0.000, C 0.000 }
gfCNCPoint2[19050] = {X 293.5330, Y 41.0522, Z -3.0000, A 0.000, B 0.000, C 0.000 }
gfCNCPoint2[19051] = {X 294.1703, Y 41.6936, Z -3.0000, A 0.000, B 0.000, C 0.000 }
gfCNCPoint2[19052] = {X 294.6516, Y 42.4590, Z -3.0000, A 0.000, B 0.000, C 0.000 }
gfCNCPoint2[19053] = {X 294.9534, Y 43.3112, Z -3.0000, A 0.000, B 0.000, C 0.000 }
gfCNCPoint2[19054] = {X 295.0611, Y 44.2089, Z -3.0000, A 0.000, B 0.000, C 0.000 }
gfCNCPoint2[19055] = {X 295.0611, Y 45.0000, Z -3.0000, A 0.000, B 0.000, C 0.000 }
gfCNCPoint2[19056] = {X 294.9608, Y 45.8901, Z -3.0000, A 0.000, B 0.000, C 0.000 }
gfCNCPoint2[19057] = {X 294.6650, Y 46.7355, Z -3.0000, A 0.000, B 0.000, C 0.000 }
gfCNCPoint2[19058] = {X 294.1885, Y 47.4940, Z -3.0000, A 0.000, B 0.000, C 0.000 }
gfCNCPoint2[19059] = {X 293.5551, Y 48.1273, Z -3.0000, A 0.000, B 0.000, C 0.000 }
gfCNCPoint2[19060] = {X 292.7967, Y 48.6039, Z -3.0000, A 0.000, B 0.000, C 0.000 }
gfCNCPoint2[19061] = {X 291.9512, Y 48.8997, Z -3.0000, A 0.000, B 0.000, C 0.000 }
gfCNCPoint2[19062] = {X 291.0611, Y 49.0000, Z -3.0000, A 0.000, B 0.000, C 0.000 }
gfCNCPoint2[19063] = {X 284.6177, Y 49.0000, Z -3.0000, A 0.000, B 0.000, C 0.000 }
gfCNCPoint2[19064] = {X 283.7276, Y 48.8997, Z -3.0000, A 0.000, B 0.000, C 0.000 }
gfCNCPoint2[19065] = {X 282.8821, Y 48.6039, Z -3.0000, A 0.000, B 0.000, C 0.000 }
gfCNCPoint2[19066] = {X 282.1237, Y 48.1273, Z -3.0000, A 0.000, B 0.000, C 0.000 }
gfCNCPoint2[19067] = {X 281.4903, Y 47.4939, Z -3.0000, A 0.000, B 0.000, C 0.000 }
gfCNCPoint2[19068] = {X 281.0138, Y 46.7355, Z -3.0000, A 0.000, B 0.000, C 0.000 }
gfCNCPoint2[19069] = {X 280.7180, Y 45.8900, Z -3.0000, A 0.000, B 0.000, C 0.000 }
gfCNCPoint2[19070] = {X 280.6177, Y 45.0000, Z -3.0000, A 0.000, B 0.000, C 0.000 }
gfCNCPoint2[19071] = {X 280.6177, Y 44.2089, Z -3.0000, A 0.000, B 0.000, C 0.000 }
gfCNCPoint2[19072] = {X 280.7232, Y 43.3126, Z -3.0000, A 0.000, B 0.000, C 0.000 }
gfCNCPoint2[19073] = {X 281.0246, Y 42.4619, Z -3.0000, A 0.000, B 0.000, C 0.000 }
gfCNCPoint2[19074] = {X 281.5068, Y 41.6991, Z -3.0000, A 0.000, B 0.000, C 0.000 }
gfCNCPoint2[19075] = {X 282.1459, Y 41.0619, Z -3.0000, A 0.000, B 0.000, C 0.000 }
gfCNCPoint2[19076] = {X 282.1457, Y 28.5928, Z -3.0000, A 0.000, B 0.000, C 0.000 }
gfCNCPoint2[19077] = {X 278.0657, Y 28.5929, Z -3.0000, A 0.000, B 0.000, C 0.000 }
gfCNCPoint2[19078] = {X 278.0657, Y 28.5929, Z 0.0000, A 0.000, B 0.000, C 0.000 }
gfCNCPoint2[19079] = {X 278.0657, Y 28.5929, Z 11.0000, A 0.000, B 0.000, C 0.000 }
gfCNCPoint2[19080] = {X 353.3541, Y 107.0430, Z 11.0000, A 0.000, B 0.000, C 0.000 }
gfCNCPoint2[19081] = {X 353.3541, Y 107.0430, Z 0.0000, A 0.000, B 0.000, C 0.000 }
gfCNCPoint2[19082] = {X 353.3541, Y 107.0430, Z -3.0000, A 0.000, B 0.000, C 0.000 }
gfCNCPoint2[19083] = {X 353.2424, Y 102.9645, Z -3.0000, A 0.000, B 0.000, C 0.000 }
gfCNCPoint2[19084] = {X 347.7202, Y 103.0331, Z -3.0000, A 0.000, B 0.000, C 0.000 }
gfCNCPoint2[19085] = {X 342.1983, Y 102.9363, Z -3.0000, A 0.000, B 0.000, C 0.000 }
gfCNCPoint2[19086] = {X 336.6819, Y 102.6744, Z -3.0000, A 0.000, B 0.000, C 0.000 }
gfCNCPoint2[19087] = {X 333.1921, Y 102.3983, Z -3.0000, A 0.000, B 0.000, C 0.000 }
gfCNCPoint2[19088] = {X 329.7159, Y 101.9854, Z -3.0000, A 0.000, B 0.000, C 0.000 }
gfCNCPoint2[19089] = {X 326.2586, Y 101.4363, Z -3.0000, A 0.000, B 0.000, C 0.000 }
gfCNCPoint2[19090] = {X 323.4092, Y 100.8313, Z -3.0000, A 0.000, B 0.000, C 0.000 }
gfCNCPoint2[19091] = {X 320.6121, Y 100.0184, Z -3.0000, A 0.000, B 0.000, C 0.000 }
gfCNCPoint2[19092] = {X 317.8823, Y 99.0020, Z -3.0000, A 0.000, B 0.000, C 0.000 }
gfCNCPoint2[19093] = {X 316.3698, Y 98.3037, Z -3.0000, A 0.000, B 0.000, C 0.000 }
gfCNCPoint2[19094] = {X 314.9207, Y 97.4817, Z -3.0000, A 0.000, B 0.000, C 0.000 }
gfCNCPoint2[19095] = {X 313.5451, Y 96.5418, Z -3.0000, A 0.000, B 0.000, C 0.000 }
gfCNCPoint2[19096] = {X 312.2527, Y 95.4905, Z -3.0000, A 0.000, B 0.000, C 0.000 }
gfCNCPoint2[19097] = {X 311.2490, Y 94.4922, Z -3.0000, A 0.000, B 0.000, C 0.000 }
gfCNCPoint2[19098] = {X 310.3707, Y 93.3819, Z -3.0000, A 0.000, B 0.000, C 0.000 }
gfCNCPoint2[19099] = {X 309.6304, Y 92.1753, Z -3.0000, A 0.000, B 0.000, C 0.000 }
gfCNCPoint2[19100] = {X 309.0385, Y 90.8893, Z -3.0000, A 0.000, B 0.000, C 0.000 }
gfCNCPoint2[19101] = {X 308.6033, Y 89.5422, Z -3.0000, A 0.000, B 0.000, C 0.000 }
gfCNCPoint2[19102] = {X 308.2598, Y 87.9191, Z -3.0000, A 0.000, B 0.000, C 0.000 }
gfCNCPoint2[19103] = {X 308.0569, Y 86.2725, Z -3.0000, A 0.000, B 0.000, C 0.000 }
gfCNCPoint2[19104] = {X 307.9960, Y 84.6146, Z -3.0000, A 0.000, B 0.000, C 0.000 }
gfCNCPoint2[19105] = {X 307.9973, Y 83.2310, Z -3.0000, A 0.000, B 0.000, C 0.000 }
gfCNCPoint2[19106] = {X 307.9973, Y 63.2123, Z -3.0000, A 0.000, B 0.000, C 0.000 }
gfCNCPoint2[19107] = {X 307.1456, Y 63.0032, Z -3.0000, A 0.000, B 0.000, C 0.000 }
gfCNCPoint2[19108] = {X 306.3538, Y 62.6265, Z -3.0000, A 0.000, B 0.000, C 0.000 }
gfCNCPoint2[19109] = {X 305.6543, Y 62.0975, Z -3.0000, A 0.000, B 0.000, C 0.000 }
gfCNCPoint2[19110] = {X 305.0760, Y 61.4382, Z -3.0000, A 0.000, B 0.000, C 0.000 }
gfCNCPoint2[19111] = {X 304.6429, Y 60.6757, Z -3.0000, A 0.000, B 0.000, C 0.000 }
gfCNCPoint2[19112] = {X 304.3726, Y 59.8414, Z -3.0000, A 0.000, B 0.000, C 0.000 }
gfCNCPoint2[19113] = {X 304.2764, Y 58.9697, Z -3.0000, A 0.000, B 0.000, C 0.000 }
gfCNCPoint2[19114] = {X 304.2762, Y 58.0000, Z -3.0000, A 0.000, B 0.000, C 0.000 }
gfCNCPoint2[19115] = {X 304.3845, Y 57.0387, Z -3.0000, A 0.000, B 0.000, C 0.000 }
gfCNCPoint2[19116] = {X 304.7040, Y 56.1256, Z -3.0000, A 0.000, B 0.000, C 0.000 }
gfCNCPoint2[19117] = {X 305.2187, Y 55.3065, Z -3.0000, A 0.000, B 0.000, C 0.000 }
gfCNCPoint2[19118] = {X 305.9027, Y 54.6225, Z -3.0000, A 0.000, B 0.000, C 0.000 }
gfCNCPoint2[19119] = {X 306.7218, Y 54.1078, Z -3.0000, A 0.000, B 0.000, C 0.000 }
gfCNCPoint2[19120] = {X 307.6349, Y 53.7883, Z -3.0000, A 0.000, B 0.000, C 0.000 }
gfCNCPoint2[19121] = {X 308.5962, Y 53.6800, Z -3.0000, A 0.000, B 0.000, C 0.000 }
gfCNCPoint2[19122] = {X 324.3107, Y 53.6800, Z -3.0000, A 0.000, B 0.000, C 0.000 }
gfCNCPoint2[19123] = {X 325.2720, Y 53.7883, Z -3.0000, A 0.000, B 0.000, C 0.000 }
gfCNCPoint2[19124] = {X 326.1851, Y 54.1078, Z -3.0000, A 0.000, B 0.000, C 0.000 }
gfCNCPoint2[19125] = {X 327.0042, Y 54.6225, Z -3.0000, A 0.000, B 0.000, C 0.000 }
gfCNCPoint2[19126] = {X 327.6882, Y 55.3065, Z -3.0000, A 0.000, B 0.000, C 0.000 }
gfCNCPoint2[19127] = {X 328.2029, Y 56.1256, Z -3.0000, A 0.000, B 0.000, C 0.000 }
gfCNCPoint2[19128] = {X 328.5224, Y 57.0387, Z -3.0000, A 0.000, B 0.000, C 0.000 }
gfCNCPoint2[19129] = {X 328.6307, Y 58.0000, Z -3.0000, A 0.000, B 0.000, C 0.000 }
gfCNCPoint2[19130] = {X 328.6307, Y 58.9360, Z -3.0000, A 0.000, B 0.000, C 0.000 }
gfCNCPoint2[19131] = {X 328.5363, Y 59.8122, Z -3.0000, A 0.000, B 0.000, C 0.000 }
gfCNCPoint2[19132] = {X 328.2677, Y 60.6515, Z -3.0000, A 0.000, B 0.000, C 0.000 }
gfCNCPoint2[19133] = {X 327.8357, Y 61.4197, Z -3.0000, A 0.000, B 0.000, C 0.000 }
gfCNCPoint2[19134] = {X 327.2581, Y 62.0852, Z -3.0000, A 0.000, B 0.000, C 0.000 }
gfCNCPoint2[19135] = {X 326.5584, Y 62.6210, Z -3.0000, A 0.000, B 0.000, C 0.000 }
gfCNCPoint2[19136] = {X 325.7653, Y 63.0051, Z -3.0000, A 0.000, B 0.000, C 0.000 }
gfCNCPoint2[19137] = {X 324.9111, Y 63.2219, Z -3.0000, A 0.000, B 0.000, C 0.000 }
gfCNCPoint2[19138] = {X 324.9126, Y 83.2296, Z -3.0000, A 0.000, B 0.000, C 0.000 }
gfCNCPoint2[19139] = {X 324.9261, Y 84.6148, Z -3.0000, A 0.000, B 0.000, C 0.000 }
gfCNCPoint2[19140] = {X 325.0035, Y 85.8501, Z -3.0000, A 0.000, B 0.000, C 0.000 }
gfCNCPoint2[19141] = {X 325.2261, Y 87.0676, Z -3.0000, A 0.000, B 0.000, C 0.000 }
gfCNCPoint2[19142] = {X 325.4715, Y 87.3365, Z -3.0000, A 0.000, B 0.000, C 0.000 }
gfCNCPoint2[19143] = {X 325.7737, Y 87.5395, Z -3.0000, A 0.000, B 0.000, C 0.000 }
gfCNCPoint2[19144] = {X 326.2239, Y 87.7938, Z -3.0000, A 0.000, B 0.000, C 0.000 }
gfCNCPoint2[19145] = {X 327.6618, Y 88.3911, Z -3.0000, A 0.000, B 0.000, C 0.000 }
gfCNCPoint2[19146] = {X 329.1568, Y 88.8266, Z -3.0000, A 0.000, B 0.000, C 0.000 }
gfCNCPoint2[19147] = {X 332.2328, Y 89.4425, Z -3.0000, A 0.000, B 0.000, C 0.000 }
gfCNCPoint2[19148] = {X 335.3453, Y 89.8352, Z -3.0000, A 0.000, B 0.000, C 0.000 }
gfCNCPoint2[19149] = {X 339.4834, Y 90.1557, Z -3.0000, A 0.000, B 0.000, C 0.000 }
gfCNCPoint2[19150] = {X 343.6300, Y 90.3354, Z -3.0000, A 0.000, B 0.000, C 0.000 }
gfCNCPoint2[19151] = {X 347.7803, Y 90.3740, Z -3.0000, A 0.000, B 0.000, C 0.000 }
gfCNCPoint2[19152] = {X 352.1620, Y 90.3356, Z -3.0000, A 0.000, B 0.000, C 0.000 }
gfCNCPoint2[19153] = {X 356.5395, Y 90.1398, Z -3.0000, A 0.000, B 0.000, C 0.000 }
gfCNCPoint2[19154] = {X 360.9071, Y 89.7867, Z -3.0000, A 0.000, B 0.000, C 0.000 }
gfCNCPoint2[19155] = {X 363.2212, Y 89.4989, Z -3.0000, A 0.000, B 0.000, C 0.000 }
gfCNCPoint2[19156] = {X 365.5139, Y 89.0725, Z -3.0000, A 0.000, B 0.000, C 0.000 }
gfCNCPoint2[19157] = {X 367.7768, Y 88.5091, Z -3.0000, A 0.000, B 0.000, C 0.000 }
gfCNCPoint2[19158] = {X 368.7089, Y 88.1958, Z -3.0000, A 0.000, B 0.000, C 0.000 }
gfCNCPoint2[19159] = {X 369.6000, Y 87.7799, Z -3.0000, A 0.000, B 0.000, C 0.000 }
gfCNCPoint2[19160] = {X 370.4387, Y 87.2667, Z -3.0000, A 0.000, B 0.000, C 0.000 }
gfCNCPoint2[19161] = {X 370.5886, Y 87.1107, Z -3.0000, A 0.000, B 0.000, C 0.000 }
gfCNCPoint2[19162] = {X 370.6659, Y 86.9086, Z -3.0000, A 0.000, B 0.000, C 0.000 }
gfCNCPoint2[19163] = {X 370.8570, Y 85.3735, Z -3.0000, A 0.000, B 0.000, C 0.000 }
gfCNCPoint2[19164] = {X 370.9208, Y 83.8280, Z -3.0000, A 0.000, B 0.000, C 0.000 }
gfCNCPoint2[19165] = {X 370.9208, Y 63.2124, Z -3.0000, A 0.000, B 0.000, C 0.000 }
gfCNCPoint2[19166] = {X 370.0691, Y 63.0034, Z -3.0000, A 0.000, B 0.000, C 0.000 }
gfCNCPoint2[19167] = {X 369.2771, Y 62.6266, Z -3.0000, A 0.000, B 0.000, C 0.000 }
gfCNCPoint2[19168] = {X 368.5775, Y 62.0977, Z -3.0000, A 0.000, B 0.000, C 0.000 }
gfCNCPoint2[19169] = {X 367.9992, Y 61.4383, Z -3.0000, A 0.000, B 0.000, C 0.000 }
gfCNCPoint2[19170] = {X 367.5660, Y 60.6758, Z -3.0000, A 0.000, B 0.000, C 0.000 }
gfCNCPoint2[19171] = {X 367.2957, Y 59.8415, Z -3.0000, A 0.000, B 0.000, C 0.000 }
gfCNCPoint2[19172] = {X 367.1994, Y 58.9697, Z -3.0000, A 0.000, B 0.000, C 0.000 }
gfCNCPoint2[19173] = {X 367.1993, Y 58.0000, Z -3.0000, A 0.000, B 0.000, C 0.000 }
gfCNCPoint2[19174] = {X 367.3076, Y 57.0387, Z -3.0000, A 0.000, B 0.000, C 0.000 }
gfCNCPoint2[19175] = {X 367.6271, Y 56.1256, Z -3.0000, A 0.000, B 0.000, C 0.000 }
gfCNCPoint2[19176] = {X 368.1418, Y 55.3065, Z -3.0000, A 0.000, B 0.000, C 0.000 }
gfCNCPoint2[19177] = {X 368.8258, Y 54.6225, Z -3.0000, A 0.000, B 0.000, C 0.000 }
gfCNCPoint2[19178] = {X 369.6449, Y 54.1078, Z -3.0000, A 0.000, B 0.000, C 0.000 }
gfCNCPoint2[19179] = {X 370.5580, Y 53.7883, Z -3.0000, A 0.000, B 0.000, C 0.000 }
gfCNCPoint2[19180] = {X 371.5193, Y 53.6800, Z -3.0000, A 0.000, B 0.000, C 0.000 }
gfCNCPoint2[19181] = {X 388.0597, Y 53.6800, Z -3.0000, A 0.000, B 0.000, C 0.000 }
gfCNCPoint2[19182] = {X 389.0210, Y 53.7883, Z -3.0000, A 0.000, B 0.000, C 0.000 }
gfCNCPoint2[19183] = {X 389.9341, Y 54.1078, Z -3.0000, A 0.000, B 0.000, C 0.000 }
gfCNCPoint2[19184] = {X 390.7532, Y 54.6225, Z -3.0000, A 0.000, B 0.000, C 0.000 }
gfCNCPoint2[19185] = {X 391.4372, Y 55.3065, Z -3.0000, A 0.000, B 0.000, C 0.000 }
gfCNCPoint2[19186] = {X 391.9519, Y 56.1256, Z -3.0000, A 0.000, B 0.000, C 0.000 }
gfCNCPoint2[19187] = {X 392.2714, Y 57.0387, Z -3.0000, A 0.000, B 0.000, C 0.000 }
gfCNCPoint2[19188] = {X 392.3797, Y 58.0000, Z -3.0000, A 0.000, B 0.000, C 0.000 }
gfCNCPoint2[19189] = {X 392.3797, Y 58.9342, Z -3.0000, A 0.000, B 0.000, C 0.000 }
gfCNCPoint2[19190] = {X 392.2645, Y 59.9250, Z -3.0000, A 0.000, B 0.000, C 0.000 }
gfCNCPoint2[19191] = {X 391.9252, Y 60.8629, Z -3.0000, A 0.000, B 0.000, C 0.000 }
gfCNCPoint2[19192] = {X 391.4817, Y 61.5731, Z -3.0000, A 0.000, B 0.000, C 0.000 }
gfCNCPoint2[19193] = {X 390.9101, Y 62.1849, Z -3.0000, A 0.000, B 0.000, C 0.000 }
gfCNCPoint2[19194] = {X 390.2316, Y 62.6757, Z -3.0000, A 0.000, B 0.000, C 0.000 }
gfCNCPoint2[19195] = {X 389.4716, Y 63.0270, Z -3.0000, A 0.000, B 0.000, C 0.000 }
gfCNCPoint2[19196] = {X 388.6583, Y 63.2260, Z -3.0000, A 0.000, B 0.000, C 0.000 }
gfCNCPoint2[19197] = {X 388.6563, Y 84.6147, Z -3.0000, A 0.000, B 0.000, C 0.000 }
gfCNCPoint2[19198] = {X 388.5965, Y 86.2731, Z -3.0000, A 0.000, B 0.000, C 0.000 }
gfCNCPoint2[19199] = {X 388.3921, Y 87.9199, Z -3.0000, A 0.000, B 0.000, C 0.000 }
gfCNCPoint2[19200] = {X 388.0448, Y 89.5426, Z -3.0000, A 0.000, B 0.000, C 0.000 }
gfCNCPoint2[19201] = {X 387.5127, Y 91.1299, Z -3.0000, A 0.000, B 0.000, C 0.000 }
gfCNCPoint2[19202] = {X 386.7632, Y 92.6269, Z -3.0000, A 0.000, B 0.000, C 0.000 }
gfCNCPoint2[19203] = {X 385.8110, Y 94.0039, Z -3.0000, A 0.000, B 0.000, C 0.000 }
gfCNCPoint2[19204] = {X 384.6752, Y 95.2338, Z -3.0000, A 0.000, B 0.000, C 0.000 }
gfCNCPoint2[19205] = {X 383.1609, Y 96.5096, Z -3.0000, A 0.000, B 0.000, C 0.000 }
gfCNCPoint2[19206] = {X 381.5198, Y 97.6174, Z -3.0000, A 0.000, B 0.000, C 0.000 }
gfCNCPoint2[19207] = {X 379.7704, Y 98.5449, Z -3.0000, A 0.000, B 0.000, C 0.000 }
gfCNCPoint2[19208] = {X 377.4992, Y 99.5010, Z -3.0000, A 0.000, B 0.000, C 0.000 }
gfCNCPoint2[19209] = {X 375.1651, Y 100.2913, Z -3.0000, A 0.000, B 0.000, C 0.000 }
gfCNCPoint2[19210] = {X 372.7802, Y 100.9116, Z -3.0000, A 0.000, B 0.000, C 0.000 }
gfCNCPoint2[19211] = {X 368.9685, Y 101.6491, Z -3.0000, A 0.000, B 0.000, C 0.000 }
gfCNCPoint2[19212] = {X 365.1257, Y 102.2024, Z -3.0000, A 0.000, B 0.000, C 0.000 }
gfCNCPoint2[19213] = {X 361.2608, Y 102.5704, Z -3.0000, A 0.000, B 0.000, C 0.000 }
gfCNCPoint2[19214] = {X 357.2538, Y 102.8111, Z -3.0000, A 0.000, B 0.000, C 0.000 }
gfCNCPoint2[19215] = {X 353.2424, Y 102.9645, Z -3.0000, A 0.000, B 0.000, C 0.000 }
gfCNCPoint2[19216] = {X 353.3519, Y 106.9630, Z -3.0000, A 0.000, B 0.000, C 0.000 }
gfCNCPoint2[19217] = {X 353.2403, Y 102.8846, Z -3.0000, A 0.000, B 0.000, C 0.000 }
gfCNCPoint2[19218] = {X 347.7204, Y 102.9531, Z -3.0000, A 0.000, B 0.000, C 0.000 }
gfCNCPoint2[19219] = {X 342.2009, Y 102.8564, Z -3.0000, A 0.000, B 0.000, C 0.000 }
gfCNCPoint2[19220] = {X 336.6868, Y 102.5946, Z -3.0000, A 0.000, B 0.000, C 0.000 }
gfCNCPoint2[19221] = {X 333.2001, Y 102.3187, Z -3.0000, A 0.000, B 0.000, C 0.000 }
gfCNCPoint2[19222] = {X 329.7269, Y 101.9062, Z -3.0000, A 0.000, B 0.000, C 0.000 }
